_CFC_ (* Continuous Function Chart, elements in execution order *)
(* set timer cycle *)
(* delay on *)
(* delay off *)
#0 hw_reset_faults_id1 <= #1.DO1
#1 PLC:PLC110_32m2(FDI1: -, FDI2: -, DI1: hw_pressure_min, DI2: hw_pressure_max, DI3: ws_pressure_min, DI4: ws_pressure_max, DI5: hw_status_alarm_id1, DI6: hw_status_alarm_id2, DI7: ws_status_alarm_id1, DI8: ws_status_alarm_id2, DI9: hw_status_run_id1, DI10: hw_status_run_id2, DI11: ws_status_run_id1, DI12: ws_status_run_id2, DI13: -, DI14: -, DI15: -, DI16: -, SI: -, status_outputs: plc_outputs)
#2 ws_output_value_id2 <= #7.ch4_value
#3 analog_inputs_module:MB110_8a(ch1_error_code: hw_error_input_pressure, ch1_value: hw_input_pressure, ch2_error_code: hw_error_output_pressure, ch2_value: hw_output_pressure, ch3_error_code: ws_error_input_pressure, ch3_value: ws_input_pressure, ch4_error_code: ws_error_output_pressure, ch4_value: ws_output_pressure, ch5_error_code: -, ch5_value: -, ch6_error_code: -, ch6_value: -, ch7_error_code: -, ch7_value: -, ch8_error_code: -, ch8_value: -, settings: #20.settings)
#4 info_analog_inputs_module <= #3.info
#5 get_aout_current_in_info(info_invertor_drive: hw_info_id_1)
#6 currents_value_pack:get_info_analog_outputs_module(ch1_current: #5, ch2_current: #85, ch3_current: #86, ch4_current: #87, ch5_current: -, ch6_current: -, ch7_current: -, ch8_current: -)
#7 analog_outputs_module:MY110_8u(info_current_channel: #6.info)
#8 hw_run_id1 <= #1.FDO1
#9 get_run_in_info(info_invertor_drive: hw_info_id_1)
#10 PLC_110_32_outputs:get_status_outputs(fdo1: #9, fdo2: #15, fdo3: #79, fdo4: #81, do1: #16, do2: #111, do3: #112, do4: #113, do5: -, do6: -, do7: -, do8: -, do9: -, do10: -, do11: -, do12: -, do13: -, do14: -, do15: -, do16: -, sdo: -)
#11 plc_outputs <= #10.get_status_outputs
#12 hw_run_id2 <= #1.FDO2
#13 ws_run_id1 <= #1.FDO3
#14 ws_run_id2 <= #1.FDO4
#15 get_run_in_info(info_invertor_drive: hw_info_id_2)
#16 get_reset_faults(info: hw_info_id_1)
#17 value_scaling(input_value: hw_output_value_id1, params_scales: out_set_frequency)
#18 hw_frequency_id1 <= #17
#19 get_params_value_scaling(in_min: 0, in_max: 1000, out_min: 0, out_max: 50)
#20 settings_channel_analog_inputs_module:SetChannelsAnalogInputsModule(ch1_ain_l: -, ch1_ain_h: -, ch1_analog_min_value: -, ch1_analog_max_value: -, ch2_ain_l: -, ch2_ain_h: -, ch2_analog_min_value: -, ch2_analog_max_value: -, ch3_ain_l: -, ch3_ain_h: -, ch3_analog_min_value: -, ch3_analog_max_value: -, ch4_ain_l: -, ch4_ain_h: -, ch4_analog_min_value: -, ch4_analog_max_value: -, ch5_ain_l: -, ch5_ain_h: -, ch5_analog_min_value: -, ch5_analog_max_value: -, ch6_ain_l: -, ch6_ain_h: -, ch6_analog_min_value: -, ch6_analog_max_value: -, ch7_ain_l: -, ch7_ain_h: -, ch7_analog_min_value: -, ch7_analog_max_value: -, ch8_ain_l: -, ch8_ain_h: -, ch8_analog_min_value: -, ch8_analog_max_value: -)
#21 plc_inputs <= #1.status_inputs
#22 get_channel_current_value(ch_number: 1, Ain_info: info_analog_inputs_module)
#23 hw_input:CurrentSensorPressure_4_20(current_value: #22, set: -)
#24 hw_input_pressure_bar <= #23.pressure
#25 hw_settings_pressure_input:SetCurrentSensorPressure_4_20(min_measure_range: hw_min_measure_range_input, max_measure_range: hw_max_measure_range_input, min_current_range: -, max_current_range: -)
#26 get_channel_current_value(ch_number: 2, Ain_info: info_analog_inputs_module)
#27 hw_output:CurrentSensorPressure_4_20(current_value: #26, set: -)
#28 ws_input:CurrentSensorPressure_4_20(current_value: #108, set: -)
#29 ws_output:CurrentSensorPressure_4_20(current_value: #109, set: -)
#30 hw_output_pressure_bar <= #27.pressure
#31 hw_settings_pressure_output:SetCurrentSensorPressure_4_20(min_measure_range: hw_min_measure_range_output, max_measure_range: hw_max_measure_range_output, min_current_range: -, max_current_range: -)
#32 ws_input_pressure_bar <= #28.pressure
#33 ws_settings_pressure_input:SetCurrentSensorPressure_4_20(min_measure_range: ws_min_measure_range_input, max_measure_range: ws_max_measure_range_input, min_current_range: -, max_current_range: -)
#34 ws_output_pressure_bar <= #29.pressure
#35 ws_settings_pressure_output:SetCurrentSensorPressure_4_20(min_measure_range: ws_min_measure_range_output, max_measure_range: ws_max_measure_range_output, min_current_range: -, max_current_range: -)
#36 hw_kpi_35:Kpi(input: #37)
#37 get_di(input_number: 1, status_inputs: plc_inputs)
#38 hw_status_run_id1_sp <= #99
#39 hw_input_low_pressure_alarm <= #36.NO
#40 hw_invertor_drive_1:InvertorDrive(start: hw_start_id_1, reset_fault: hw_id1_reset_faults, low_pressure_in: #36.NO, high_pressure_out: #75.NO, status_run: #99, status_alarm: #46, ain_value: hw_output_pressure_bar, aout_value: hw_frequency_id_1, auto: hw_id1_auto, direct_logic: -, set_point: hw_set_point_pressure, P: -, I: -, D: -, manual: hw_manual_set_frequency_id1, min_range: -, max_range: -, active: hw_id1_active, system_alarm: hw_alarm_on)
#41 pid1:PID(#43.actual, #43.set_point, #43.P, #43.I, #43.D, #43.Y_manual, #43.Y_offset, #43.Y_min, #43.Y_max, #43.manual, #41.out 3)
#42 hw_info_id_1 <= #40.info
#43 hw_settings_pid_id_1:params_in_set_PID(set: #40.settings_pid)
#44 hw_frequency_id_1 <= #41.out 1
#45 get_di(input_number: 2, status_inputs: plc_inputs)
#46 get_di(input_number: 5, status_inputs: plc_inputs)
#47 hw_invertor_drive_2:InvertorDrive(start: hw_start_id_2, reset_fault: hw_id2_reset_faults, low_pressure_in: #36.NO, high_pressure_out: #75.NO, status_run: #101, status_alarm: #100, ain_value: hw_output_pressure_bar, aout_value: hw_frequency_id_2, auto: hw_id2_auto, direct_logic: -, set_point: hw_set_point_pressure, P: -, I: -, D: -, manual: hw_manual_set_frequency_id2, min_range: -, max_range: -, active: hw_id2_active, system_alarm: hw_alarm_on)
#48 pid2:PID(#49.actual, #49.set_point, #49.P, #49.I, #49.D, #49.Y_manual, #49.Y_offset, #49.Y_min, #49.Y_max, #49.manual, #48.out 3)
#49 hw_settings_pid_id_2:params_in_set_PID(set: #47.settings_pid)
#50 hw_frequency_id_2 <= #48.out 1
#51 get_di(input_number: 3, status_inputs: plc_inputs)
#52 hw_status_run_id2_sp <= #101
#53 ws_invertor_drive_1:InvertorDrive(start: ws_start_id_1, reset_fault: ws_id1_reset_faults, low_pressure_in: #58.NO, high_pressure_out: #76.NO, status_run: #104, status_alarm: #103, ain_value: ws_output_pressure_bar, aout_value: ws_frequency_id_1, auto: ws_id1_auto, direct_logic: -, set_point: ws_set_point_pressure, P: -, I: -, D: -, manual: ws_manual_set_frequency_id1, min_range: -, max_range: -, active: ws_id1_active, system_alarm: ws_alarm_on)
#54 pid3:PID(#56.actual, #56.set_point, #56.P, #56.I, #56.D, #56.Y_manual, #56.Y_offset, #56.Y_min, #56.Y_max, #56.manual, #54.out 3)
#55 ws_info_id_1 <= #53.info
#56 ws_settings_pid_id_1:params_in_set_PID(set: #53.settings_pid)
#57 ws_frequency_id_1 <= #54.out 1
#58 ws_kpi_35:Kpi(input: #51)
#59 ws_invertor_drive_2:InvertorDrive(start: ws_start_id_2, reset_fault: ws_id2_reset_faults, low_pressure_in: #58.NO, high_pressure_out: #76.NO, status_run: #107, status_alarm: #105, ain_value: ws_output_pressure_bar, aout_value: ws_frequency_id_2, auto: ws_id2_auto, direct_logic: -, set_point: ws_set_point_pressure, P: -, I: -, D: -, manual: ws_manual_set_frequency_id2, min_range: -, max_range: -, active: ws_id2_active, system_alarm: ws_alarm_on)
#60 pid4:PID(#62.actual, #62.set_point, #62.P, #62.I, #62.D, #62.Y_manual, #62.Y_offset, #62.Y_min, #62.Y_max, #62.manual, #60.out 3)
#61 ws_info_id_2 <= #59.info
#62 ws_settings_pid_id_2:params_in_set_PID(set: #59.settings_pid)
#63 ws_frequency_id_2 <= #60.out 1
#64 ws_status_run_id1_sp <= #104
#65 hw_single_mode:Single(enable: hw_single_enable, pivot_pump: hw_pivot_single, info_invertor_drive1: hw_info_id_1, info_invertor_drive2: hw_info_id_2, info_invertor_drive3: -, info_invertor_drive4: -, info_invertor_drive5: -, info_invertor_drive6: -, info_invertor_drive7: -, info_invertor_drive8: -)
#66 hw_mode_selector:Cascade_Cycle_Selector(cascade: hw_cascade_enable, cycle: hw_cycle_enable, single: hw_single_enable, info_single: #65.info_single, info_cycle: #69.info_cycle, info_cascade: #70.info_cascade)
#67 hw_start_id_1 <= #66.start_pump1
#68 hms_to_time(hours: hw_cycle_set_hours, minutes: hw_cycle_set_minutes, seconds: hw_cycle_set_seconds)
#69 hw_cycle_mode:cycle(enable: hw_cycle_enable, set_timer: #68, info_invertor_drive1: hw_info_id_1, info_invertor_drive2: hw_info_id_2, info_invertor_drive3: -, info_invertor_drive4: -, info_invertor_drive5: -, info_invertor_drive6: -, info_invertor_drive7: -, info_invertor_drive8: -)
#70 hw_cascade_mode:cascade(enable: hw_cascade_enable, set_pressure: hw_set_point_pressure, in_pressure: hw_input_pressure_bar, pivot_pump: hw_pivot_cascade, delay_on: #72, delay_off: #73, info_invertor_drive1: hw_info_id_1, info_invertor_drive2: hw_info_id_2, info_invertor_drive3: -, info_invertor_drive4: -, info_invertor_drive5: -, info_invertor_drive6: -, info_invertor_drive7: -, info_invertor_drive8: -)
#71 hw_start_id_2 <= #66.start_pump2
#72 hms_to_time(hours: hw_cascade_delay_on_hours, minutes: hw_cascade_delay_on_minutes, seconds: hw_cascade_delay_on_seconds)
#73 hms_to_time(hours: hw_cascade_delay_off_hours, minutes: hw_cascade_delay_off_minutes, seconds: hw_cascade_delay_off_seconds)
#74 hw_info_id_2 <= #47.info
#75 hw_kpi_36:Kpi(input: #45)
#76 ws_kpi_36:Kpi(input: #102)
#77 hw_reset_faults_id2 <= #1.DO2
#78 ws_reset_faults_id1 <= #1.DO3
#79 get_run_in_info(info_invertor_drive: ws_info_id_1)
#80 ws_reset_faults_id2 <= #1.DO4
#81 get_run_in_info(info_invertor_drive: ws_info_id_2)
#82 hw_output_value_id1 <= #7.ch1_value
#83 hw_output_value_id2 <= #7.ch2_value
#84 ws_output_value_id1 <= #7.ch3_value
#85 get_aout_current_in_info(info_invertor_drive: hw_info_id_2)
#86 get_aout_current_in_info(info_invertor_drive: ws_info_id_1)
#87 get_aout_current_in_info(info_invertor_drive: ws_info_id_2)
(* set timer cycle *)
(* delay on *)
(* delay off *)
#88 ws_single_mode:Single(enable: ws_single_enable, pivot_pump: ws_pivot_single, info_invertor_drive1: ws_info_id_1, info_invertor_drive2: ws_info_id_2, info_invertor_drive3: -, info_invertor_drive4: -, info_invertor_drive5: -, info_invertor_drive6: -, info_invertor_drive7: -, info_invertor_drive8: -)
#89 ws_mode_selector:Cascade_Cycle_Selector(cascade: ws_cascade_enable, cycle: ws_cycle_enable, single: ws_single_enable, info_single: #88.info_single, info_cycle: #93.info_cycle, info_cascade: #94.info_cascade)
#90 ws_start_id_1 <= #89.start_pump1
#91 hw_mode_error <= #66.mode_selector_error
#92 hms_to_time(hours: ws_cycle_set_hours, minutes: ws_cycle_set_minutes, seconds: ws_cycle_set_seconds)
#93 ws_cycle_mode:cycle(enable: ws_cycle_enable, set_timer: #92, info_invertor_drive1: ws_info_id_1, info_invertor_drive2: ws_info_id_2, info_invertor_drive3: -, info_invertor_drive4: -, info_invertor_drive5: -, info_invertor_drive6: -, info_invertor_drive7: -, info_invertor_drive8: -)
#94 ws_cascade_mode:cascade(enable: ws_cascade_enable, set_pressure: ws_set_point_pressure, in_pressure: ws_input_pressure_bar, pivot_pump: ws_pivot_cascade, delay_on: #97, delay_off: #98, info_invertor_drive1: ws_info_id_1, info_invertor_drive2: ws_info_id_2, info_invertor_drive3: -, info_invertor_drive4: -, info_invertor_drive5: -, info_invertor_drive6: -, info_invertor_drive7: -, info_invertor_drive8: -)
#95 ws_mode_error <= #89.mode_selector_error
#96 ws_start_id_2 <= #89.start_pump2
#97 hms_to_time(hours: ws_cascade_delay_on_hours, minutes: ws_cascade_delay_on_minutes, seconds: ws_cascade_delay_on_seconds)
#98 hms_to_time(hours: ws_cascade_delay_off_hours, minutes: ws_cascade_delay_off_minutes, seconds: ws_cascade_delay_off_seconds)
#99 get_di(input_number: 9, status_inputs: plc_inputs)
#100 get_di(input_number: 6, status_inputs: plc_inputs)
#101 get_di(input_number: 10, status_inputs: plc_inputs)
#102 get_di(input_number: 4, status_inputs: plc_inputs)
#103 get_di(input_number: 7, status_inputs: plc_inputs)
#104 get_di(input_number: 11, status_inputs: plc_inputs)
#105 get_di(input_number: 8, status_inputs: plc_inputs)
#106 ws_input_low_pressure_alarm <= #58.NO
#107 get_di(input_number: 12, status_inputs: plc_inputs)
#108 get_channel_current_value(ch_number: 3, Ain_info: info_analog_inputs_module)
#109 get_channel_current_value(ch_number: 4, Ain_info: info_analog_inputs_module)
#110 out_set_frequency <= #19
#111 get_reset_faults(info: hw_info_id_2)
#112 get_reset_faults(info: ws_info_id_1)
#113 get_reset_faults(info: ws_info_id_2)
#114 ws_status_run_id2_sp <= #107
#115 hw_out_high_pressure_alarm <= #75.NO
#116 ws_input_low_pressure_alarm <= #76.NO
#117 value_scaling(input_value: hw_output_value_id2, params_scales: out_set_frequency)
#118 hw_frequency_id2 <= #117
#119 value_scaling(input_value: ws_output_value_id1, params_scales: out_set_frequency)
#120 ws_frequency_id1 <= #119
#121 value_scaling(input_value: ws_output_value_id2, params_scales: out_set_frequency)
#122 ws_frequency_id2 <= #121
#123 get_di(input_number: 1, status_inputs: plc_inputs)
#124 get_di(input_number: 2, status_inputs: plc_inputs)
#125 hw_alarm_manager:ALARM_MANAGER(low_pressure_input: #123, high_pressure_out: #124, external_alarm_invertor_drive_code: #135.error_code_alarm, input_pressure_error_code: hw_error_input_pressure, out_pressure_error_code: hw_error_output_pressure, mode_selector_error: hw_mode_error)
#126 hw_alarm_on <= #125.alarm_on
#127 hw_alarm_error_code <= #125.error_code_alarm
#128 hw_alarm_message <= #125.error_message
#129 get_di(input_number: 3, status_inputs: plc_inputs)
#130 get_di(input_number: 4, status_inputs: plc_inputs)
#131 hw_alarm_manager:ALARM_MANAGER(low_pressure_input: #129, high_pressure_out: #130, external_alarm_invertor_drive_code: #136.error_code_alarm, input_pressure_error_code: ws_error_input_pressure, out_pressure_error_code: ws_error_output_pressure, mode_selector_error: ws_mode_error)
#132 ws_alarm_on <= #131.alarm_on
#133 ws_alarm_error_code <= #131.error_code_alarm
#134 ws_alarm_message <= #131.error_message
#135 hw_external_alarm:external_alarm_invertor_drive(status_inputs: plc_inputs, number_di_alarm_id1: 5, number_di_alarm_id2: 6, number_di_alarm_id3: -, number_di_alarm_id4: -, number_di_alarm_id5: -, number_di_alarm_id6: -, number_di_alarm_id7: -, number_di_alarm_id8: -)
#136 ws_external_alarm:external_alarm_invertor_drive(status_inputs: plc_inputs, number_di_alarm_id1: 7, number_di_alarm_id2: 8, number_di_alarm_id3: -, number_di_alarm_id4: -, number_di_alarm_id5: -, number_di_alarm_id6: -, number_di_alarm_id7: -, number_di_alarm_id8: -)
_END_CFC_
END_PROGRAM

(* POU PLC110_32/PLC110_32m2, ST *)
FUNCTION_BLOCK PLC110_32m2

VAR_INPUT
	FDI1:BOOL;
	FDI2:BOOL;
	DI1:BOOL;
	DI2:BOOL;
	DI3:BOOL;
	DI4:BOOL;
	DI5:BOOL;
	DI6:BOOL;
	DI7:BOOL;
	DI8:BOOL;
	DI9:BOOL;
	DI10:BOOL;
	DI11:BOOL;
	DI12:BOOL;
	DI13:BOOL;
	DI14:BOOL;
	DI15:BOOL;
	DI16:BOOL;
	SI:BOOL;
	status_outputs:classPLC32m2StatusOutputs;
END_VAR

VAR_OUTPUT
	FDO1:BOOL;
	FDO2:BOOL;
	FDO3:BOOL;
	FDO4:BOOL;
	DO1:BOOL;
	DO2:BOOL;
	DO3:BOOL;
	DO4:BOOL;
	DO5:BOOL;
	DO6:BOOL;
	DO7:BOOL;
	DO8:BOOL;
	DO9:BOOL;
	DO10:BOOL;
	DO11:BOOL;
	DO12:BOOL;
	DO13:BOOL;
	DO14:BOOL;
	DO15:BOOL;
	DO16:BOOL;
	SO:BOOL;
	status_inputs:classPLC32m2StatusInputs;
END_VAR

VAR
	fast_inputs:classFastDiscreteInputs;
	discrete_inputs:classDiscreteInputs;
	special_input:classSpecialInput;
	fast_outputs:classFastDiscreteOutputs;
	discrete_outputs:classDiscreteOutputs;
	special_output:classSpecialOutput;
END_VAR
init;

get_status_inputs;

get_status_outputs;
END_FUNCTION_BLOCK
ACTION get_status_inputs:
status_inputs.fast_inputs:=fast_inputs;
status_inputs.discrete_inputs:=discrete_inputs;
status_inputs.special_input:=special_input;
END_ACTION
ACTION get_status_outputs:
FDO1:=status_outputs.fast_outputs.Bit1;
FDO2:=status_outputs.fast_outputs.Bit2;
FDO3:=status_outputs.fast_outputs.Bit3;
FDO4:=status_outputs.fast_outputs.Bit4;

DO1:=status_outputs.discrete_outputs.first_byte.Bit1;
DO2:=status_outputs.discrete_outputs.first_byte.Bit2;
DO3:=status_outputs.discrete_outputs.first_byte.Bit3;
DO4:=status_outputs.discrete_outputs.first_byte.Bit4;
DO5:=status_outputs.discrete_outputs.first_byte.Bit5;
DO6:=status_outputs.discrete_outputs.first_byte.Bit6;
DO7:=status_outputs.discrete_outputs.first_byte.Bit7;
DO8:=status_outputs.discrete_outputs.first_byte.Bit8;
DO9:=status_outputs.discrete_outputs.second_byte.Bit1;
DO10:=status_outputs.discrete_outputs.second_byte.Bit2;
DO11:=status_outputs.discrete_outputs.second_byte.Bit3;
DO12:=status_outputs.discrete_outputs.second_byte.Bit4;
DO13:=status_outputs.discrete_outputs.second_byte.Bit5;
DO14:=status_outputs.discrete_outputs.second_byte.Bit6;
DO15:=status_outputs.discrete_outputs.second_byte.Bit7;
DO16:=status_outputs.discrete_outputs.second_byte.Bit8;

SO:=status_outputs.special_output.Bit1;
END_ACTION
ACTION init:
fast_inputs.Bit1:=FDI1;
fast_inputs.Bit2:=FDI2;

discrete_inputs.first_byte.Bit1:=DI1;
discrete_inputs.first_byte.Bit2:=DI2;
discrete_inputs.first_byte.Bit3:=DI3;
discrete_inputs.first_byte.Bit4:=DI4;
discrete_inputs.first_byte.Bit5:=DI5;
discrete_inputs.first_byte.Bit6:=DI6;
discrete_inputs.first_byte.Bit7:=DI7;
discrete_inputs.first_byte.Bit8:=DI8;
discrete_inputs.second_byte.Bit1:=DI9;
discrete_inputs.second_byte.Bit2:=DI10;
discrete_inputs.second_byte.Bit3:=DI11;
discrete_inputs.second_byte.Bit4:=DI12;
discrete_inputs.second_byte.Bit5:=DI13;
discrete_inputs.second_byte.Bit6:=DI14;
discrete_inputs.second_byte.Bit7:=DI15;
discrete_inputs.second_byte.Bit8:=DI16;

special_input.Bit1:=SI;

fast_outputs.Bit1:=FDO1;
fast_outputs.Bit2:=FDO2;
fast_outputs.Bit3:=FDO3;
fast_outputs.Bit4:=FDO4;

discrete_outputs.first_byte.Bit1:=DO1;
discrete_outputs.first_byte.Bit2:=DO2;
discrete_outputs.first_byte.Bit3:=DO3;
discrete_outputs.first_byte.Bit4:=DO4;
discrete_outputs.first_byte.Bit5:=DO5;
discrete_outputs.first_byte.Bit6:=DO6;
discrete_outputs.first_byte.Bit7:=DO7;
discrete_outputs.first_byte.Bit8:=DO8;

discrete_outputs.second_byte.Bit1:=DO9;
discrete_outputs.second_byte.Bit2:=DO10;
discrete_outputs.second_byte.Bit3:=DO11;
discrete_outputs.second_byte.Bit4:=DO12;
discrete_outputs.second_byte.Bit5:=DO13;
discrete_outputs.second_byte.Bit6:=DO14;
discrete_outputs.second_byte.Bit7:=DO15;
discrete_outputs.second_byte.Bit8:=DO16;

special_output.Bit1:=SO;
END_ACTION

(* POU PLC110_32/get_status_outputs, ST *)
FUNCTION_BLOCK get_status_outputs

VAR_INPUT
	fdo1:BOOL:=FALSE;
	fdo2:BOOL:=FALSE;
	fdo3:BOOL:=FALSE;
	fdo4:BOOL:=FALSE;
	do1:BOOL:=FALSE;
	do2:BOOL:=FALSE;
	do3:BOOL:=FALSE;
	do4:BOOL:=FALSE;
	do5:BOOL:=FALSE;
	do6:BOOL:=FALSE;
	do7:BOOL:=FALSE;
	do8:BOOL:=FALSE;
	do9:BOOL:=FALSE;
	do10:BOOL:=FALSE;
	do11:BOOL:=FALSE;
	do12:BOOL:=FALSE;
	do13:BOOL:=FALSE;
	do14:BOOL:=FALSE;
	do15:BOOL:=FALSE;
	do16:BOOL:=FALSE;
	sdo:BOOL:=FALSE;
END_VAR

VAR_OUTPUT
	get_status_outputs:classPLC32m2StatusOutputs;
END_VAR
get_status_outputs := get_status_outputs_def(fdo1, fdo2, fdo3, fdo4, do1, do2, do3, do4, do5, do6, do7, do8, do9, do10, do11, do12, do13, do14, do15, do16, sdo);
END_FUNCTION_BLOCK

(* POU PLC110_32/get_status_outputs_def, ST *)
FUNCTION get_status_outputs_def : classPLC32m2StatusOutputs

VAR_INPUT
	fdo1:BOOL:=FALSE;
	fdo2:BOOL:=FALSE;
	fdo3:BOOL:=FALSE;
	fdo4:BOOL:=FALSE;
	do1:BOOL:=FALSE;
	do2:BOOL:=FALSE;
	do3:BOOL:=FALSE;
	do4:BOOL:=FALSE;
	do5:BOOL:=FALSE;
	do6:BOOL:=FALSE;
	do7:BOOL:=FALSE;
	do8:BOOL:=FALSE;
	do9:BOOL:=FALSE;
	do10:BOOL:=FALSE;
	do11:BOOL:=FALSE;
	do12:BOOL:=FALSE;
	do13:BOOL:=FALSE;
	do14:BOOL:=FALSE;
	do15:BOOL:=FALSE;
	do16:BOOL:=FALSE;
	sdo:BOOL:=FALSE;
END_VAR
get_status_outputs_def.fast_outputs.Bit1:=fdo1;
get_status_outputs_def.fast_outputs.Bit2:=fdo2;
get_status_outputs_def.fast_outputs.Bit3:=fdo3;
get_status_outputs_def.fast_outputs.Bit4:=fdo4;

get_status_outputs_def.discrete_outputs.first_byte.Bit1:=do1;
get_status_outputs_def.discrete_outputs.first_byte.Bit2:=do2;
get_status_outputs_def.discrete_outputs.first_byte.Bit3:=do3;
get_status_outputs_def.discrete_outputs.first_byte.Bit4:=do4;
get_status_outputs_def.discrete_outputs.first_byte.Bit5:=do5;
get_status_outputs_def.discrete_outputs.first_byte.Bit6:=do6;
get_status_outputs_def.discrete_outputs.first_byte.Bit7:=do7;
get_status_outputs_def.discrete_outputs.first_byte.Bit8:=do8;
get_status_outputs_def.discrete_outputs.second_byte.Bit1:=do9;
get_status_outputs_def.discrete_outputs.second_byte.Bit2:=do10;
get_status_outputs_def.discrete_outputs.second_byte.Bit3:=do11;
get_status_outputs_def.discrete_outputs.second_byte.Bit4:=do12;
get_status_outputs_def.discrete_outputs.second_byte.Bit5:=do13;
get_status_outputs_def.discrete_outputs.second_byte.Bit6:=do14;
get_status_outputs_def.discrete_outputs.second_byte.Bit7:=do15;
get_status_outputs_def.discrete_outputs.second_byte.Bit8:=do16;

get_status_outputs_def.special_output.Bit1:=sdo;
END_FUNCTION

(* POU MB110_8.A/MB110_8a, ST *)
FUNCTION_BLOCK MB110_8a

VAR_INPUT
	ch1_error_code:WORD:=61447;
	ch1_value:REAL;
	ch2_error_code:WORD:=61447;
	ch2_value:REAL;
	ch3_error_code:WORD:=61447;
	ch3_value:REAL;
	ch4_error_code:WORD:=61447;
	ch4_value:REAL;
	ch5_error_code:WORD:=61447;
	ch5_value:REAL;
	ch6_error_code:WORD:=61447;
	ch6_value:REAL;
	ch7_error_code:WORD:=61447;
	ch7_value:REAL;
	ch8_error_code:WORD:=61447;
	ch8_value:REAL;
	settings:classSetAnalogInputsModule;
END_VAR

VAR_OUTPUT
	info:classInfoAnalogInputModule;
END_VAR
get_info_message;
END_FUNCTION_BLOCK
ACTION get_info_message:
info.channel1.error_message:=get_error_code(ch1_error_code);
info.channel2.error_message:=get_error_code(ch2_error_code);
info.channel3.error_message:=get_error_code(ch3_error_code);
info.channel4.error_message:=get_error_code(ch4_error_code);
info.channel5.error_message:=get_error_code(ch5_error_code);
info.channel6.error_message:=get_error_code(ch6_error_code);
info.channel7.error_message:=get_error_code(ch7_error_code);
info.channel8.error_message:=get_error_code(ch8_error_code);

info.channel1.current_value:=get_current_value(ch1_error_code,settings.ch1_set, ch1_value);
info.channel2.current_value:=get_current_value(ch2_error_code,settings.ch2_set, ch2_value);
info.channel3.current_value:=get_current_value(ch3_error_code,settings.ch3_set, ch3_value);
info.channel4.current_value:=get_current_value(ch4_error_code,settings.ch4_set, ch4_value);
info.channel5.current_value:=get_current_value(ch5_error_code,settings.ch5_set, ch5_value);
info.channel6.current_value:=get_current_value(ch6_error_code,settings.ch6_set, ch6_value);
info.channel7.current_value:=get_current_value(ch7_error_code,settings.ch7_set, ch7_value);
info.channel8.current_value:=get_current_value(ch8_error_code,settings.ch8_set, ch8_value);
END_ACTION

(* POU MB110_8.A/get_error_code, ST *)
FUNCTION get_error_code: STRING(79)
(* ï¿½ï¿½ï¿½ï¿½ï¿½ï¿½ï¿½ ï¿½ï¿½ï¿½ï¿½ï¿½ï¿½ï¿½ï¿½ï¿½ï¿½ï¿½ï¿½ï¿½ï¿½ ï¿½ï¿½ï¿½ï¿½ ï¿½ï¿½ï¿½ï¿½ï¿½ï¿½ ï¿½ï¿½ï¿½ï¿½ï¿½ï¿½ï¿½ï¿½ ï¿½ï¿½ï¿½ï¿½ï¿½ï¿½ï¿½ï¿½ï¿½ï¿½ï¿½ ï¿½ï¿½ï¿½ï¿½ï¿½ï¿½ ï¿½ï¿½ï¿½ï¿½ï¿½ï¿½ *)

VAR_INPUT
	code_error: WORD;
END_VAR

VAR
	error_message: STRING(79);
END_VAR
IF code_error=0
	THEN error_message := 'ï¿½ï¿½ï¿½ï¿½ï¿½ï¿½ï¿½ï¿½ï¿½ ï¿½ï¿½ï¿½ï¿½ï¿½ï¿½ï¿½';
ELSIF code_error = 61440
	THEN error_message := 'ï¿½ï¿½ï¿½ï¿½ï¿½ï¿½ï¿½ï¿½ ï¿½ï¿½ï¿½ï¿½ï¿½ï¿½ï¿½ï¿½ ï¿½ï¿½ï¿½ï¿½ï¿½ï¿½ï¿½';
ELSIF code_error = 61446
	THEN error_message := 'ï¿½ï¿½ï¿½ï¿½ï¿½ï¿½ ï¿½ï¿½ ï¿½ï¿½ï¿½ï¿½ï¿½ï¿½. ï¿½ï¿½ï¿½ï¿½ï¿½ ï¿½ï¿½ï¿½ï¿½ï¿½ï¿½ï¿½ï¿½ï¿½ï¿½ï¿½ ï¿½ï¿½ï¿½ï¿½ï¿½ï¿½ï¿½ ï¿½ï¿½ï¿½ï¿½ï¿½ï¿½ï¿½ï¿½ï¿½.';
ELSIF code_error = 61447
	THEN error_message := 'ï¿½ï¿½ï¿½ï¿½ï¿½ï¿½ ï¿½ï¿½ï¿½ï¿½ï¿½ï¿½ï¿½ï¿½.';
ELSIF code_error = 61448
	THEN error_message := 'ï¿½ï¿½ï¿½ï¿½ï¿½ï¿½ ï¿½ï¿½ï¿½ï¿½ï¿½ï¿½ï¿½ï¿½ï¿½ï¿½ï¿½ ï¿½ï¿½ï¿½ï¿½ï¿½ï¿½ï¿½ï¿½ï¿½ ï¿½ï¿½ï¿½ï¿½ï¿½ï¿½ ï¿½ï¿½.';
ELSIF code_error = 61449
	THEN error_message := 'ï¿½ï¿½ï¿½ï¿½ ï¿½ï¿½ï¿½ï¿½ï¿½ï¿½ï¿½ï¿½ï¿½ï¿½ï¿½ ï¿½ï¿½ï¿½ï¿½ï¿½ï¿½ï¿½ï¿½ï¿½ ï¿½ï¿½ï¿½ï¿½ï¿½ï¿½ ï¿½ï¿½.';
ELSIF code_error = 61450
	THEN error_message := 'ï¿½ï¿½ï¿½ï¿½ï¿½ï¿½ï¿½ï¿½ï¿½ï¿½ ï¿½ï¿½ï¿½ï¿½ï¿½ï¿½ï¿½ï¿½ ï¿½ï¿½ï¿½ï¿½ï¿½ï¿½ï¿½ ï¿½ï¿½ï¿½ï¿½ï¿½ï¿½.';
ELSIF code_error = 61451
	THEN error_message := 'ï¿½ï¿½ï¿½ï¿½ï¿½ï¿½ï¿½ï¿½ï¿½ï¿½ ï¿½ï¿½ï¿½ï¿½ï¿½ï¿½ï¿½ï¿½ ï¿½ï¿½ï¿½ï¿½ï¿½ï¿½ï¿½ ï¿½ï¿½ï¿½ï¿½.';
ELSIF code_error = 61452
	THEN error_message := 'ï¿½ï¿½ï¿½ï¿½ï¿½ï¿½ï¿½ï¿½ ï¿½ï¿½ï¿½ï¿½ï¿½ï¿½ï¿½ï¿½ï¿½ ï¿½ï¿½ï¿½ï¿½ï¿½ï¿½ï¿½.';
ELSIF code_error = 61453
	THEN error_message := 'ï¿½ï¿½ï¿½ï¿½ï¿½ ï¿½ï¿½ï¿½ï¿½ï¿½ï¿½ï¿½.';
ELSIF code_error = 61454
	THEN error_message := 'ï¿½ï¿½ï¿½ï¿½ï¿½ï¿½ï¿½ï¿½ï¿½ï¿½ ï¿½ï¿½ï¿½ï¿½ï¿½ ï¿½ ï¿½ï¿½ï¿½.';
ELSIF code_error = 61455
	THEN error_message := 'ï¿½ï¿½ï¿½ï¿½ï¿½ï¿½ï¿½ï¿½ï¿½ï¿½ï¿½ï¿½ ï¿½ï¿½ï¿½ï¿½ï¿½ï¿½ï¿½ï¿½ï¿½ï¿½ï¿½ï¿½ï¿½ ï¿½ï¿½ï¿½ï¿½ï¿½ï¿½ï¿½ï¿½ï¿½ï¿½ï¿½.';
ELSE
	error_message := 'Error not Found';
END_IF

get_error_code := error_message;
END_FUNCTION

(* POU MB110_8.A/get_current_value, ST *)
FUNCTION get_current_value : REAL
(* ï¿½ï¿½ï¿½ï¿½ï¿½ï¿½ï¿½ ï¿½ï¿½ï¿½ï¿½ï¿½ï¿½ï¿½ï¿½ï¿½ï¿½ï¿½ï¿½ï¿½ï¿½ï¿½ ï¿½ï¿½ï¿½ï¿½ï¿½ï¿½ ï¿½ ï¿½ï¿½ï¿½ ï¿½ ï¿½ï¿½ï¿½ï¿½ï¿½ï¿½ï¿½ï¿½ ï¿½ï¿½ï¿½ï¿½ *)

VAR_INPUT
	code_error:WORD;
	ch_set:classSetAnalogInputChannel;
	ch_value:REAL;
END_VAR
IF code_error = 0 THEN
	get_current_value := value_scaling(ch_value, get_set_Ain_value_params(ch_set));
ELSE
	(* ï¿½ï¿½ï¿½ï¿½ ï¿½ï¿½ï¿½ï¿½ï¿½ï¿½ ï¿½ï¿½ï¿½ï¿½ï¿½ï¿½ ï¿½ï¿½ï¿½ï¿½ï¿½ï¿½ ï¿½ï¿½ï¿½ï¿½ï¿½ï¿½ï¿½ ï¿½ï¿½ï¿½ï¿½ï¿½ï¿½ *)
	get_current_value := -8;
END_IF;
END_FUNCTION

(* POU function/value_scale/value_scaling, ST *)
FUNCTION value_scaling : REAL
(* ï¿½ï¿½ï¿½ï¿½ï¿½ï¿½ï¿½ ï¿½ï¿½ï¿½ï¿½ï¿½ï¿½ï¿½ï¿½ï¿½ï¿½ï¿½ï¿½ï¿½ï¿½ï¿½ ï¿½ï¿½ï¿½ï¿½ï¿½ *)

VAR_INPUT
	input_value: REAL;
	params_scales:classParamsValueScaling;
END_VAR

VAR
	A: REAL;
	B: REAL;
END_VAR
A := (params_scales.out_max - params_scales.out_min) / (params_scales.in_max - params_scales.in_min);
B := ((params_scales.out_min * params_scales.in_max) - (params_scales.out_max * params_scales.in_min)) / (params_scales.in_max - params_scales.in_min);

value_scaling := A * input_value + B;
END_FUNCTION

(* POU MB110_8.A/get_set_Ain_value_params, ST *)
FUNCTION get_set_Ain_value_params : classParamsValueScaling
(* ï¿½ï¿½ï¿½ï¿½ï¿½ï¿½ï¿½ï¿½ï¿½ï¿½ï¿½ï¿½ï¿½ï¿½ ï¿½ï¿½ ï¿½ï¿½ï¿½ï¿½ ï¿½ï¿½ï¿½ï¿½ï¿½ï¿½ï¿½ï¿½ ï¿½ï¿½ï¿½ï¿½ï¿½ ï¿½ ï¿½ï¿½ï¿½ï¿½ï¿½ï¿½ï¿½ï¿½ï¿½ ï¿½ï¿½ï¿½ï¿½ï¿½ï¿½ï¿½ï¿½ï¿½ï¿½ï¿½ï¿½ï¿½ï¿½ï¿½ *)

VAR_INPUT
	set:classSetAnalogInputChannel;
END_VAR
get_set_Ain_value_params.in_min:=set.ain_l;
get_set_Ain_value_params.in_max:=set.ain_h;
get_set_Ain_value_params.out_min:=set.analog_min_value;
get_set_Ain_value_params.out_max:=set.analog_max_value;
END_FUNCTION

(* POU MB110_8U/get_info_analog_outputs_module, ST *)
FUNCTION_BLOCK get_info_analog_outputs_module

VAR_INPUT
	ch1_current:REAL;
	ch2_current:REAL;
	ch3_current:REAL;
	ch4_current:REAL;
	ch5_current:REAL;
	ch6_current:REAL;
	ch7_current:REAL;
	ch8_current:REAL;
END_VAR

VAR_OUTPUT
	info:classAnalogOutputModule;
END_VAR
info.channel1.current_value := ch1_current;
info.channel2.current_value := ch2_current;
info.channel3.current_value := ch3_current;
info.channel4.current_value := ch4_current;
info.channel5.current_value := ch5_current;
info.channel6.current_value := ch6_current;
info.channel7.current_value := ch7_current;
info.channel8.current_value := ch8_current;
END_FUNCTION_BLOCK

(* POU MB110_8U/MY110_8u, ST *)
FUNCTION_BLOCK MY110_8u

VAR_INPUT
	info_current_channel:classAnalogOutputModule;
END_VAR

VAR_OUTPUT
	ch1_value:WORD;
	ch2_value:WORD;
	ch3_value:WORD;
	ch4_value:WORD;
	ch5_value:WORD;
	ch6_value:WORD;
	ch7_value:WORD;
	ch8_value:WORD;
END_VAR

VAR
	ch_ain_l: REAL := 4;  (* ï¿½ï¿½ï¿½ï¿½ï¿½ï¿½ï¿½ï¿½ ï¿½ï¿½ï¿½ï¿½ï¿½ï¿½ ï¿½ï¿½ï¿½ï¿½ï¿½ï¿½ï¿½ ï¿½ï¿½ï¿½ï¿½ï¿½ï¿½ï¿½ï¿½ ï¿½ï¿½ï¿½ï¿½ï¿½ï¿½ï¿½ï¿½ï¿½ *)
	ch_ain_h: REAL := 20;  (* ï¿½ï¿½ï¿½ï¿½ï¿½ï¿½ï¿½ï¿½ ï¿½ï¿½ï¿½ï¿½ï¿½ï¿½ï¿½ ï¿½ï¿½ï¿½ï¿½ï¿½ï¿½ï¿½ ï¿½ï¿½ï¿½ï¿½ï¿½ï¿½ï¿½ï¿½ ï¿½ï¿½ï¿½ï¿½ï¿½ï¿½ï¿½ï¿½ï¿½ *)
	ch_analog_min_value: REAL :=  0;  (* ï¿½ï¿½ï¿½ï¿½ï¿½ï¿½ ï¿½ï¿½ï¿½ï¿½ï¿½ï¿½ï¿½ ï¿½ï¿½ï¿½ *)
	ch_analog_max_value: REAL := 1000;  (* ï¿½ï¿½ï¿½ï¿½ï¿½ï¿½ï¿½ ï¿½ï¿½ï¿½ï¿½ï¿½ï¿½ï¿½ ï¿½ï¿½ï¿½ *)
	set_params:classParamsValueScaling;
END_VAR
set_params := get_params_value_scaling(ch_ain_l, ch_ain_h, ch_analog_min_value, ch_analog_max_value);

ch1_value := REAL_TO_INT(value_scaling(info_current_channel.channel1.current_value, set_params));
ch2_value := REAL_TO_INT(value_scaling(info_current_channel.channel2.current_value, set_params));
ch3_value := REAL_TO_INT(value_scaling(info_current_channel.channel3.current_value, set_params));
ch4_value := REAL_TO_INT(value_scaling(info_current_channel.channel4.current_value, set_params));
ch5_value := REAL_TO_INT(value_scaling(info_current_channel.channel5.current_value, set_params));
ch6_value := REAL_TO_INT(value_scaling(info_current_channel.channel6.current_value, set_params));
ch7_value := REAL_TO_INT(value_scaling(info_current_channel.channel7.current_value, set_params));
ch8_value := REAL_TO_INT(value_scaling(info_current_channel.channel8.current_value, set_params));
END_FUNCTION_BLOCK

(* POU function/value_scale/get_params_value_scaling, ST *)
FUNCTION get_params_value_scaling : classParamsValueScaling

VAR_INPUT
	in_min: REAL;
	in_max: REAL;
	out_min: REAL;
	out_max: REAL;
END_VAR
get_params_value_scaling.in_min := in_min;
get_params_value_scaling.in_max := in_max;
get_params_value_scaling.out_min := out_min;
get_params_value_scaling.out_max := out_max;
END_FUNCTION

(* POU MB110_8.A/SetChannelsAnalogInputsModule, ST *)
FUNCTION_BLOCK SetChannelsAnalogInputsModule

VAR_INPUT
	(* ï¿½ï¿½ï¿½ï¿½ï¿½ï¿½ï¿½ï¿½ï¿½ï¿½ï¿½ï¿½ï¿½ï¿½ï¿½ï¿½ ï¿½ï¿½ï¿½ï¿½ï¿½ï¿½ï¿½ï¿½ï¿½ ï¿½ï¿½ï¿½ï¿½ï¿½ï¿½ ï¿½ï¿½ï¿½ï¿½ï¿½ï¿½. ï¿½ï¿½. ï¿½ï¿½ï¿½ï¿½ï¿½ï¿½ï¿½ï¿½ï¿½ï¿½ ï¿½ï¿½ï¿½ï¿½ï¿½ï¿½ï¿½: ï¿½ï¿½ï¿½ï¿½ï¿½ï¿½ï¿½ï¿½ï¿½ï¿½. ï¿½ï¿½ï¿½ï¿½ï¿½ï¿½ï¿½ ï¿½.2 *)
	(* ï¿½ï¿½ï¿½ï¿½ï¿½ï¿½ï¿½ ï¿½ï¿½ï¿½ ï¿½ ï¿½ï¿½ï¿½ï¿½ï¿½ï¿½ï¿½ï¿½ ï¿½ï¿½ ï¿½ï¿½ï¿½ï¿½ï¿½ï¿½ï¿½ï¿½ï¿½: ï¿½ï¿½ï¿½ ï¿½ï¿½ï¿½ï¿½ï¿½ï¿½ï¿½ 4-20mA  *)

	ch1_ain_l: REAL := 0;  (* ï¿½ï¿½ï¿½ï¿½ï¿½ï¿½ï¿½ï¿½ Ain.L *)
	ch1_ain_h: REAL := 100;  (* ï¿½ï¿½ï¿½ï¿½ï¿½ï¿½ï¿½ï¿½ Ain.H *)
	ch1_analog_min_value: REAL := 4;  (* ï¿½ï¿½ï¿½ï¿½ï¿½ï¿½ï¿½ï¿½ ï¿½ï¿½ï¿½ï¿½ï¿½ï¿½ ï¿½ï¿½ï¿½ï¿½ï¿½ï¿½ï¿½ ï¿½ï¿½ï¿½ï¿½ï¿½ï¿½ï¿½ *)
	ch1_analog_max_value: REAL := 20;  (* ï¿½ï¿½ï¿½ï¿½ï¿½ï¿½ï¿½ï¿½ ï¿½ï¿½ï¿½ï¿½ï¿½ï¿½ï¿½ ï¿½ï¿½ï¿½ï¿½ï¿½ï¿½ï¿½ ï¿½ï¿½ï¿½ï¿½ï¿½ï¿½ï¿½ *)

	ch2_ain_l: REAL := 0;  (* ï¿½ï¿½ï¿½ï¿½ï¿½ï¿½ï¿½ï¿½ Ain.L *)
	ch2_ain_h: REAL := 100;  (* ï¿½ï¿½ï¿½ï¿½ï¿½ï¿½ï¿½ï¿½ Ain.H *)
	ch2_analog_min_value: REAL := 4;  (* ï¿½ï¿½ï¿½ï¿½ï¿½ï¿½ï¿½ï¿½ ï¿½ï¿½ï¿½ï¿½ï¿½ï¿½ ï¿½ï¿½ï¿½ï¿½ï¿½ï¿½ï¿½ ï¿½ï¿½ï¿½ï¿½ï¿½ï¿½ï¿½ *)
	ch2_analog_max_value: REAL := 20;  (* ï¿½ï¿½ï¿½ï¿½ï¿½ï¿½ï¿½ï¿½ ï¿½ï¿½ï¿½ï¿½ï¿½ï¿½ï¿½ ï¿½ï¿½ï¿½ï¿½ï¿½ï¿½ï¿½ ï¿½ï¿½ï¿½ï¿½ï¿½ï¿½ï¿½ *)

	ch3_ain_l: REAL := 0;  (* ï¿½ï¿½ï¿½ï¿½ï¿½ï¿½ï¿½ï¿½ Ain.L *)
	ch3_ain_h: REAL := 100;  (* ï¿½ï¿½ï¿½ï¿½ï¿½ï¿½ï¿½ï¿½ Ain.H *)
	ch3_analog_min_value: REAL := 4;  (* ï¿½ï¿½ï¿½ï¿½ï¿½ï¿½ï¿½ï¿½ ï¿½ï¿½ï¿½ï¿½ï¿½ï¿½ ï¿½ï¿½ï¿½ï¿½ï¿½ï¿½ï¿½ ï¿½ï¿½ï¿½ï¿½ï¿½ï¿½ï¿½ *)
	ch3_analog_max_value: REAL := 20;  (* ï¿½ï¿½ï¿½ï¿½ï¿½ï¿½ï¿½ï¿½ ï¿½ï¿½ï¿½ï¿½ï¿½ï¿½ï¿½ ï¿½ï¿½ï¿½ï¿½ï¿½ï¿½ï¿½ ï¿½ï¿½ï¿½ï¿½ï¿½ï¿½ï¿½ *)

	ch4_ain_l: REAL := 0;  (* ï¿½ï¿½ï¿½ï¿½ï¿½ï¿½ï¿½ï¿½ Ain.L *)
	ch4_ain_h: REAL := 100;  (* ï¿½ï¿½ï¿½ï¿½ï¿½ï¿½ï¿½ï¿½ Ain.H *)
	ch4_analog_min_value: REAL := 4;  (* ï¿½ï¿½ï¿½ï¿½ï¿½ï¿½ï¿½ï¿½ ï¿½ï¿½ï¿½ï¿½ï¿½ï¿½ ï¿½ï¿½ï¿½ï¿½ï¿½ï¿½ï¿½ ï¿½ï¿½ï¿½ï¿½ï¿½ï¿½ï¿½ *)
	ch4_analog_max_value: REAL := 20;  (* ï¿½ï¿½ï¿½ï¿½ï¿½ï¿½ï¿½ï¿½ ï¿½ï¿½ï¿½ï¿½ï¿½ï¿½ï¿½ ï¿½ï¿½ï¿½ï¿½ï¿½ï¿½ï¿½ ï¿½ï¿½ï¿½ï¿½ï¿½ï¿½ï¿½ *)

	ch5_ain_l: REAL := 0;  (* ï¿½ï¿½ï¿½ï¿½ï¿½ï¿½ï¿½ï¿½ Ain.L *)
	ch5_ain_h: REAL := 100;  (* ï¿½ï¿½ï¿½ï¿½ï¿½ï¿½ï¿½ï¿½ Ain.H *)
	ch5_analog_min_value: REAL := 4;  (* ï¿½ï¿½ï¿½ï¿½ï¿½ï¿½ï¿½ï¿½ ï¿½ï¿½ï¿½ï¿½ï¿½ï¿½ ï¿½ï¿½ï¿½ï¿½ï¿½ï¿½ï¿½ ï¿½ï¿½ï¿½ï¿½ï¿½ï¿½ï¿½ *)
	ch5_analog_max_value: REAL := 20;  (* ï¿½ï¿½ï¿½ï¿½ï¿½ï¿½ï¿½ï¿½ ï¿½ï¿½ï¿½ï¿½ï¿½ï¿½ï¿½ ï¿½ï¿½ï¿½ï¿½ï¿½ï¿½ï¿½ ï¿½ï¿½ï¿½ï¿½ï¿½ï¿½ï¿½ *)

	ch6_ain_l: REAL := 0;  (* ï¿½ï¿½ï¿½ï¿½ï¿½ï¿½ï¿½ï¿½ Ain.L *)
	ch6_ain_h: REAL := 100;  (* ï¿½ï¿½ï¿½ï¿½ï¿½ï¿½ï¿½ï¿½ Ain.H *)
	ch6_analog_min_value: REAL := 4;  (* ï¿½ï¿½ï¿½ï¿½ï¿½ï¿½ï¿½ï¿½ ï¿½ï¿½ï¿½ï¿½ï¿½ï¿½ ï¿½ï¿½ï¿½ï¿½ï¿½ï¿½ï¿½ ï¿½ï¿½ï¿½ï¿½ï¿½ï¿½ï¿½ *)
	ch6_analog_max_value: REAL := 20;  (* ï¿½ï¿½ï¿½ï¿½ï¿½ï¿½ï¿½ï¿½ ï¿½ï¿½ï¿½ï¿½ï¿½ï¿½ï¿½ ï¿½ï¿½ï¿½ï¿½ï¿½ï¿½ï¿½ ï¿½ï¿½ï¿½ï¿½ï¿½ï¿½ï¿½ *)

	ch7_ain_l: REAL := 0;  (* ï¿½ï¿½ï¿½ï¿½ï¿½ï¿½ï¿½ï¿½ Ain.L *)
	ch7_ain_h: REAL := 100;  (* ï¿½ï¿½ï¿½ï¿½ï¿½ï¿½ï¿½ï¿½ Ain.H *)
	ch7_analog_min_value: REAL := 4;  (* ï¿½ï¿½ï¿½ï¿½ï¿½ï¿½ï¿½ï¿½ ï¿½ï¿½ï¿½ï¿½ï¿½ï¿½ ï¿½ï¿½ï¿½ï¿½ï¿½ï¿½ï¿½ ï¿½ï¿½ï¿½ï¿½ï¿½ï¿½ï¿½ *)
	ch7_analog_max_value: REAL := 20;  (* ï¿½ï¿½ï¿½ï¿½ï¿½ï¿½ï¿½ï¿½ ï¿½ï¿½ï¿½ï¿½ï¿½ï¿½ï¿½ ï¿½ï¿½ï¿½ï¿½ï¿½ï¿½ï¿½ ï¿½ï¿½ï¿½ï¿½ï¿½ï¿½ï¿½ *)

	ch8_ain_l: REAL := 0;  (* ï¿½ï¿½ï¿½ï¿½ï¿½ï¿½ï¿½ï¿½ Ain.L *)
	ch8_ain_h: REAL := 100;  (* ï¿½ï¿½ï¿½ï¿½ï¿½ï¿½ï¿½ï¿½ Ain.H *)
	ch8_analog_min_value: REAL := 4;  (* ï¿½ï¿½ï¿½ï¿½ï¿½ï¿½ï¿½ï¿½ ï¿½ï¿½ï¿½ï¿½ï¿½ï¿½ ï¿½ï¿½ï¿½ï¿½ï¿½ï¿½ï¿½ ï¿½ï¿½ï¿½ï¿½ï¿½ï¿½ï¿½ *)
	ch8_analog_max_value: REAL := 20;  (* ï¿½ï¿½ï¿½ï¿½ï¿½ï¿½ï¿½ï¿½ ï¿½ï¿½ï¿½ï¿½ï¿½ï¿½ï¿½ ï¿½ï¿½ï¿½ï¿½ï¿½ï¿½ï¿½ ï¿½ï¿½ï¿½ï¿½ï¿½ï¿½ï¿½ *)
END_VAR

VAR_OUTPUT
	settings:classSetAnalogInputsModule;
END_VAR
get_settings;
END_FUNCTION_BLOCK
ACTION get_settings:
settings.ch1_set := get_setAin(ch1_ain_l, ch1_ain_h, ch1_analog_min_value, ch1_analog_max_value);
settings.ch2_set := get_setAin(ch2_ain_l, ch2_ain_h, ch2_analog_min_value, ch2_analog_max_value);
settings.ch3_set := get_setAin(ch3_ain_l, ch3_ain_h, ch3_analog_min_value, ch3_analog_max_value);
settings.ch4_set := get_setAin(ch4_ain_l, ch4_ain_h, ch4_analog_min_value, ch4_analog_max_value);
settings.ch5_set := get_setAin(ch5_ain_l, ch5_ain_h, ch5_analog_min_value, ch5_analog_max_value);
settings.ch6_set := get_setAin(ch6_ain_l, ch6_ain_h, ch6_analog_min_value, ch6_analog_max_value);
settings.ch7_set := get_setAin(ch7_ain_l, ch7_ain_h, ch7_analog_min_value, ch7_analog_max_value);
settings.ch8_set := get_setAin(ch8_ain_l, ch8_ain_h, ch8_analog_min_value, ch8_analog_max_value);
END_ACTION

(* POU MB110_8.A/get_setAin, ST *)
FUNCTION get_setAin : classSetAnalogInputChannel
(* ï¿½ï¿½ï¿½ï¿½ï¿½ï¿½ï¿½ï¿½ï¿½ ï¿½ï¿½ï¿½ï¿½ï¿½ï¿½ï¿½ï¿½ ï¿½ dataclass *)

VAR_INPUT
	ch_ain_l: REAL := 0;  (* ï¿½ï¿½ï¿½ï¿½ï¿½ï¿½ï¿½ï¿½ Ain.L *)
	ch_ain_h: REAL := 100;  (* ï¿½ï¿½ï¿½ï¿½ï¿½ï¿½ï¿½ï¿½ Ain.H *)
	ch_analog_min_value: REAL := 4;  (* ï¿½ï¿½ï¿½ï¿½ï¿½ï¿½ï¿½ï¿½ ï¿½ï¿½ï¿½ï¿½ï¿½ï¿½ ï¿½ï¿½ï¿½ï¿½ï¿½ï¿½ï¿½ ï¿½ï¿½ï¿½ï¿½ï¿½ï¿½ï¿½ *)
	ch_analog_max_value: REAL := 20;  (* ï¿½ï¿½ï¿½ï¿½ï¿½ï¿½ï¿½ï¿½ ï¿½ï¿½ï¿½ï¿½ï¿½ï¿½ï¿½ ï¿½ï¿½ï¿½ï¿½ï¿½ï¿½ï¿½ ï¿½ï¿½ï¿½ï¿½ï¿½ï¿½ï¿½ *)
END_VAR
get_setAin.ain_l:=ch_ain_l;
get_setAin.ain_h:=ch_ain_h;
get_setAin.analog_min_value:=ch_analog_min_value;
get_setAin.analog_max_value:=ch_analog_max_value;
END_FUNCTION

(* POU PressureSensor_4_20ma/CurrentSensorPressure_4_20, ST *)
FUNCTION_BLOCK CurrentSensorPressure_4_20

VAR_INPUT
	current_value:REAL;  (*ï¿½ï¿½ï¿½ï¿½ï¿½ï¿½ï¿½ï¿½ ï¿½ï¿½ï¿½ï¿½ 4-20ï¿½ï¿½ *)
	set:classSetPressureSensor4_20;  (* ï¿½ï¿½ï¿½ï¿½ï¿½ï¿½ï¿½ ï¿½ ï¿½ï¿½ï¿½ï¿½ï¿½ï¿½ ï¿½ï¿½ï¿½ï¿½ï¿½ï¿½ï¿½ ï¿½ï¿½ï¿½ï¿½ï¿½ï¿½ï¿½ï¿½ *)
END_VAR

VAR_OUTPUT
	pressure:REAL;  (* ï¿½ï¿½ï¿½ï¿½ï¿½ï¿½ï¿½ï¿½ ï¿½ï¿½ ï¿½ï¿½ï¿½ï¿½ï¿½ï¿½ *)
END_VAR
pressure:=value_scaling(current_value, get_set_sensor_value_params(set));
END_FUNCTION_BLOCK

(* POU PressureSensor_4_20ma/get_set_sensor_value_params, ST *)
FUNCTION get_set_sensor_value_params : classParamsValueScaling

VAR_INPUT
	sensor_set:classSetPressureSensor4_20;
END_VAR
get_set_sensor_value_params.in_min := sensor_set.min_current_range;
get_set_sensor_value_params.in_max := sensor_set.max_current_range;
get_set_sensor_value_params.out_min := sensor_set.min_measure_range;
get_set_sensor_value_params.out_max := sensor_set.max_measure_range;
END_FUNCTION

(* POU Invertor_Drive/InvertorDrive, ST *)
FUNCTION_BLOCK InvertorDrive
(* Function block implementation invertor drive. *)

VAR_INPUT
(* discrete inputs *)
	start: BOOL := FALSE;
	reset_fault: BOOL := FALSE;
	low_pressure_in: BOOL;  (* external alarm *)
	high_pressure_out: BOOL;  (* external alrm *)
(* discrete outputs *)
	status_run: BOOL;
	status_alarm: BOOL;
(* analog inputs *)
	ain_value: REAL := 0;  (* mA or V *)
(* analog outputs *)
	aout_value: REAL := 0;
(* PID settings *)
	auto: BOOL := FALSE;
	direct_logic: BOOL := TRUE;  (* flag forward/reverse control, reverse control: if input value less set point, output value to less. forward control: if input value less set point, output value to more. *)
	set_point: REAL := 0;  (* set point, measure system in input value control. *)
	P: REAL := 2;  (* proporcional value of PID, if more, out value fasted. *)
	I: INT := 10;  (* integral value of PID, seconds *)
	D:INT := 0;  (* differential value PID, seconds *)

(* limit work frequency *)
	manual: REAL := 0; (* set output value in manual mode, Hz*)
	min_range: REAL := 15;  (* min value in manual mode, Hz*)
	max_range: REAL := 50;  (* max value in manual mode, Hz*)

(* status invertor in work *)
	active: BOOL := FALSE;  (* statis active invertor drive. *)
	system_alarm: BOOL; (* alarm manager alarm_on *)
END_VAR

VAR_OUTPUT
	info: classInfoInvertorDrive;
	settings_pid: classSetPid;
END_VAR

VAR
	invertor_drive: classInvertorDrive;
    set_auto: classSetAutoInvertorDrive;
	set_frequency: classSetLimitFrequency;
	set_pid: classSetPid;

	discrete_inputs: classInvertorDriveDiscreteInputs;
	discrete_outputs: classInvertorDriveDiscreteOutputs;
	analog_inputs: classInvertorDriveAnalogInputs;
	analog_outputs: classInvertorDriveAnalogOutputs;

	overflow: BOOL := FALSE; (* overflow integral value of PID *)

	external_alarm:STRING(79); (* message of external alarm. *)

	info_alarm: classAlarmInvertorDrive;
END_VAR
init;

info_alarm.external_alarm := get_external_alarm(
	discrete_inputs.low_pressure_in, discrete_inputs.high_pressure_out
);

get_PID_set;

get_infomessage;
END_FUNCTION_BLOCK
ACTION get_infoMessage:
info.active := active;
info.set_pid := set_pid;
info.alarm.external_alarm := info_alarm.external_alarm;

IF discrete_outputs.status_alarm THEN
	info_alarm.fault_invertor_drive := 'Alarm invertor drive!';
	analog_outputs.out_frequency := 0;
ELSE
	info_alarm.fault_invertor_drive := 'No alarm';
END_IF;

info.alarm.fault_invertor_drive := info_alarm.fault_invertor_drive;

IF discrete_outputs.status_run THEN
	info.status_run := 'Run';

ELSE
	info.status_run := 'Stopped';
	analog_outputs.out_frequency := 0;
END_IF;

(* converted frequency in current value of 4-20 mA *)
info.frequency := analog_outputs.out_frequency;
info.aout_frequency := value_scaling(analog_outputs.out_frequency, get_params_value_scaling(0, 50, 4, 20));

IF info.alarm.external_alarm  <> 'GOOD' THEN
	discrete_inputs.start := FALSE;
ELSIF info.alarm.fault_invertor_drive <> 'No alarm' THEN
	discrete_inputs.start := FALSE;
ELSIF system_alarm <> 0 THEN
	discrete_inputs.start := FALSE;
ELSE
	discrete_inputs.start := invertor_drive.discrete_inputs.start;
END_IF;

info.reset_fault := discrete_inputs.reset_fault;

info.run := discrete_inputs.start;
END_ACTION
ACTION get_PID_set:
analog_inputs := invertor_drive.analog_input;
set_auto := invertor_drive.set.set_auto;
set_frequency := invertor_drive.set.set_frequency;

overflow := FALSE; (* this place for realise reset integral value of PID *) 

set_pid := get_set_pid(
	set_auto.direct_logic,
	set_auto.value,
	set_auto.set_point,
	set_auto.P,
	set_auto.I,
	set_auto.D,
	set_frequency.manual,
	0,
	set_frequency.min_range,
	set_frequency.max_range,
	NOT set_auto.auto,
	overflow
);

settings_pid := set_pid;
END_ACTION
ACTION init:
invertor_drive.analog_input.set_frequency := ain_value;
invertor_drive.analog_output.out_frequency := aout_value;

invertor_drive.discrete_inputs.start := start;
invertor_drive.discrete_inputs.reset_fault := reset_fault;
invertor_drive.discrete_inputs.low_pressure_in := low_pressure_in;
invertor_drive.discrete_inputs.high_pressure_out := high_pressure_out;

invertor_drive.discrete_outputs.status_run := status_run;
invertor_drive.discrete_outputs.status_alarm := status_alarm;

invertor_drive.set.set_frequency.min_range := min_range;
invertor_drive.set.set_frequency.max_range := max_range;

invertor_drive.set.set_auto.auto := auto;
invertor_drive.set.set_auto.direct_logic := direct_logic;
invertor_drive.set.set_auto.set_point := set_point;
invertor_drive.set.set_auto.value := ain_value;
invertor_drive.set.set_auto.P := P;
invertor_drive.set.set_auto.I := I;
invertor_drive.set.set_auto.D := D;

invertor_drive.set.set_frequency.manual := manual;
invertor_drive.set.set_frequency.min_range := min_range;
invertor_drive.set.set_frequency.max_range := max_range;

discrete_inputs := invertor_drive.discrete_inputs;
discrete_outputs := invertor_drive.discrete_outputs;
analog_outputs := invertor_drive.analog_output;
END_ACTION

(* POU Invertor_Drive/get_external_alarm, ST *)
FUNCTION get_external_alarm : STRING(79)
(* ï¿½ï¿½ï¿½ï¿½ï¿½ï¿½ï¿½ï¿½ï¿½ ï¿½ï¿½ï¿½ï¿½ï¿½ï¿½ï¿½ï¿½ï¿½ ï¿½ï¿½ï¿½ï¿½ï¿½ï¿½ ï¿½ï¿½ ï¿½ï¿½ï¿½ï¿½ï¿½ï¿½ ï¿½ï¿½ï¿½ï¿½ ï¿½ï¿½ï¿½ ï¿½ï¿½ï¿½ï¿½ï¿½ï¿½ï¿½ï¿½ï¿½ï¿½ ï¿½ï¿½ï¿½ï¿½ï¿½ï¿½ï¿½ï¿½ *)
VAR_INPUT
	low_pressure_in:BOOL;
	high_pressure_out:BOOL;
END_VAR
IF low_pressure_in THEN
	get_external_alarm:='ï¿½ï¿½ï¿½ï¿½ï¿½ï¿½ ï¿½ï¿½ï¿½ï¿½ï¿½ï¿½ï¿½ï¿½ ï¿½ï¿½ ï¿½ï¿½ï¿½ï¿½ï¿½';
ELSIF high_pressure_out THEN
	get_external_alarm:='ï¿½ï¿½ï¿½ï¿½ï¿½ï¿½ï¿½ ï¿½ï¿½ï¿½ï¿½ï¿½ï¿½ï¿½ï¿½ ï¿½ï¿½ ï¿½ï¿½ï¿½ï¿½ï¿½ï¿½';
ELSE
	get_external_alarm:='GOOD';
END_IF;
END_FUNCTION

(* POU PID_regulator/get_set_pid, ST *)
FUNCTION get_set_pid : classSetPid

VAR_INPUT
	direct_logic:BOOL:=TRUE;
	actual:REAL;
	set_point:REAL;
	P:REAL:=2;  (* ï¿½ï¿½ï¿½ï¿½ï¿½ï¿½ï¿½ï¿½ï¿½ï¿½ï¿½ï¿½ï¿½ï¿½ï¿½ï¿½ ï¿½ï¿½ï¿½ï¿½ï¿½ï¿½ï¿½ï¿½ï¿½ï¿½ï¿½ ï¿½ï¿½ï¿½ï¿½ï¿½ï¿½ï¿½ï¿½ï¿½ï¿½, ï¿½ï¿½ï¿½ ï¿½ï¿½ï¿½ï¿½ï¿½ï¿½ï¿½ï¿½ï¿½ï¿½ ï¿½ï¿½ï¿½ï¿½ï¿½ ï¿½ï¿½ï¿½ï¿½ï¿½ï¿½ï¿½ï¿½ï¿½ï¿½ ï¿½ï¿½ï¿½ï¿½ï¿½ï¿½ï¿½ï¿½ï¿½ï¿½ ï¿½ï¿½ï¿½ï¿½ï¿½ï¿½ï¿½*)
	I:INT:=10;  (* ï¿½ï¿½ï¿½ï¿½ï¿½ï¿½ï¿½ï¿½ï¿½ï¿½ï¿½ï¿½ ï¿½ï¿½ï¿½ï¿½ï¿½ï¿½ï¿½ï¿½ï¿½ï¿½ï¿½ ï¿½ï¿½ï¿½ï¿½ï¿½ï¿½ï¿½ï¿½ï¿½ï¿½, ï¿½ï¿½ï¿½ï¿½ï¿½ ï¿½ ï¿½ï¿½ï¿½ï¿½ï¿½ï¿½ï¿½ï¿½ *)
	D:INT:=0;  (* ï¿½ï¿½ï¿½ï¿½ï¿½ï¿½ï¿½ï¿½ï¿½ï¿½ï¿½ï¿½ï¿½ï¿½ï¿½ï¿½ ï¿½ï¿½ï¿½ï¿½ï¿½ï¿½ï¿½ï¿½ï¿½ï¿½ï¿½ ï¿½ï¿½ï¿½ï¿½ï¿½ï¿½ï¿½ï¿½ï¿½ï¿½, ï¿½ï¿½ï¿½ï¿½ï¿½ ï¿½ ï¿½ï¿½ï¿½ï¿½ï¿½ï¿½ï¿½ï¿½ *)
	Y_manual:REAL:=0;  (* Hz *)
	Y_offset:REAL:=0;
	Y_min:REAL;
	Y_max:REAL;
	manual:BOOL:=TRUE;  (* ï¿½ï¿½ï¿½ï¿½ï¿½ï¿½ï¿½ï¿½ï¿½ï¿½ï¿½ ï¿½ï¿½ï¿½ï¿½ï¿½ï¿½ï¿½ï¿½ ï¿½ï¿½ï¿½ï¿½ï¿½ï¿½ ï¿½ï¿½ï¿½ï¿½ï¿½ *)
	reset:BOOL:=FALSE;
END_VAR
IF direct_logic = TRUE THEN
	get_set_pid.actual := actual;
	get_set_pid.set_point := set_point;
ELSE
	get_set_pid.actual := set_point;
	get_set_pid.set_point := actual;
END_IF;

get_set_pid.P := P;
get_set_pid.I := I;
get_set_pid.D := D;
get_set_pid.Y_manual := Y_manual;
get_set_pid.Y_offset := Y_offset;
get_set_pid.Y_min := Y_min;
get_set_pid.Y_max := Y_max;
get_set_pid.manual := manual;
get_set_pid.reset := reset;
END_FUNCTION

(* POU PID_regulator/params_in_set_PID, ST *)
FUNCTION_BLOCK params_in_set_PID

VAR_INPUT
	set:classSetPid;
END_VAR

VAR_OUTPUT
	actual:REAL;
	set_point:REAL;
	P:REAL;
	I:REAL;
	D:REAL;
	Y_manual:REAL;
	Y_offset:REAL;
	Y_min:REAL;
	Y_max:REAL;
	manual:BOOL;
	reset:BOOL;
END_VAR
actual := set.actual;
set_point := set.set_point;
P := set.P;
I := set.I;
D := set.D;
Y_manual := set.Y_manual;
Y_offset := set.Y_offset;
Y_min := set.Y_min;
Y_max := set.Y_max;
manual := set.manual;
reset := set.reset;
END_FUNCTION_BLOCK

(* POU single_mode/Single, ST *)
FUNCTION_BLOCK Single
(* Function block implementation single mode. *)

VAR_INPUT
    enable: BOOL; (* Enable single mode *)
    pivot_pump: INT; (* pivot pump *)
    info_invertor_drive1: classInfoInvertorDrive;
    info_invertor_drive2: classInfoInvertorDrive;
    info_invertor_drive3: classInfoInvertorDrive;
    info_invertor_drive4: classInfoInvertorDrive;
    info_invertor_drive5: classInfoInvertorDrive;
    info_invertor_drive6: classInfoInvertorDrive;
    info_invertor_drive7: classInfoInvertorDrive;
    info_invertor_drive8: classInfoInvertorDrive;
END_VAR

VAR_OUTPUT
    info_single: classInfoSingle; (* info mode *)
END_VAR

VAR
    pivot: INT;
    pumps: ARRAY[1..8] OF BOOL;
END_VAR
pumps[1] := get_active(info_invertor_drive1);
pumps[2] := get_active(info_invertor_drive2);
pumps[3] := get_active(info_invertor_drive3);
pumps[4] := get_active(info_invertor_drive4);
pumps[5] := get_active(info_invertor_drive5);
pumps[6] := get_active(info_invertor_drive6);
pumps[7] := get_active(info_invertor_drive7);
pumps[8] := get_active(info_invertor_drive8);

pivot := pivot_pump;
IF pivot = 0 THEN
	enable := FALSE;
    info_single.error_code:=8;
END_IF;

IF enable THEN
    IF pumps[pivot] THEN
        info_single.pivot_pump := pivot;
        info_single.start_pump := pumps[pivot];
        info_single.error_code := 0;
        info_single.message := 'Select pump in work'; (* Выбранный насос в работе. *)
    ELSE
        info_single.pivot_pump := -8;
        info_single.start_pump := FALSE;
        info_single.error_code := 6;
        info_single.message := 'Select pump is not active!'; (* Выбранный насос не активен! *)
    END_IF;
      
ELSE
    info_single.pivot_pump := -8;
    info_single.start_pump := FALSE;
    info_single.error_code := 8;
    info_single.message := 'Single mode is not activate'; (* Режим работы одного насоса не активен. *)
END_IF;
END_FUNCTION_BLOCK

(* POU Invertor_Drive/get_active, ST *)
FUNCTION get_active : BOOL

VAR_INPUT
	info_invertor_drive:classInfoInvertorDrive;
END_VAR
get_active:=info_invertor_drive.active;
END_FUNCTION

(* POU cycle_mode/cycle, ST *)
FUNCTION_BLOCK cycle
(* Function block implementation cycle mode. *)

VAR_INPUT
	enable:BOOL;
	set_timer:TIME;
	info_invertor_drive1: classInfoInvertorDrive;
    info_invertor_drive2: classInfoInvertorDrive;
    info_invertor_drive3: classInfoInvertorDrive;
    info_invertor_drive4: classInfoInvertorDrive;
    info_invertor_drive5: classInfoInvertorDrive;
    info_invertor_drive6: classInfoInvertorDrive;
    info_invertor_drive7: classInfoInvertorDrive;
    info_invertor_drive8: classInfoInvertorDrive;
	END_VAR

VAR_OUTPUT
	info_cycle:classInfoCycle;
END_VAR
VAR
	pumps: ARRAY [1..8] OF BOOL;
	i: INT := 8;
	start_timer: TIME:=t#0ms;
	start_delay:TON;
	in: BOOL;

	working_time:TIME;
	Q:BOOL;
	n: INT;
END_VAR
pumps[1] := get_active(info_invertor_drive1);
pumps[2] := get_active(info_invertor_drive2);
pumps[3] := get_active(info_invertor_drive3);
pumps[4] := get_active(info_invertor_drive4);
pumps[5] := get_active(info_invertor_drive5);
pumps[6] := get_active(info_invertor_drive6);
pumps[7] := get_active(info_invertor_drive7);
pumps[8] := get_active(info_invertor_drive8);

n:=i;

IF pumps[i] = FALSE THEN
	i := i + 1;
END_IF;

IF  start_timer = t#0ms THEN
	start_timer := get_systime();
	in := TRUE;
END_IF;

working_time := work_time(start_timer);


IF working_time >= set_timer THEN
	in := FALSE;
	i := i + 1;
	start_timer := t#0ms;
END_IF;

start_delay(IN:=in, PT:=t#3s);
Q := start_delay.Q;

IF i > 8 THEN
	i := 1;
END_IF;

IF enable THEN
	info_cycle.working_time := working_time;
	info_cycle.run_timer := Q;
	info_cycle.pump_number := n;
ELSE
	info_cycle.working_time := T#0s;
	info_cycle.run_timer := FALSE;
	info_cycle.pump_number := 1;
	start_timer := t#0s;
END_IF;
info_cycle.error_code := 0;
END_FUNCTION_BLOCK

(* POU cycle_mode/get_systime, ST *)
FUNCTION get_systime : TIME

VAR_INPUT
END_VAR
get_systime:=TIME();
END_FUNCTION

(* POU cycle_mode/work_time, ST *)
FUNCTION work_time : TIME

VAR_INPUT
	start:TIME;
END_VAR
work_time:=TIME() - start;
END_FUNCTION

(* POU cascade_mode/cascade, ST *)
FUNCTION_BLOCK cascade
(* Functional block implementation cascade mode. *)
VAR_INPUT
	enable:BOOL;
	set_pressure:REAL;
	in_pressure: REAL;
	pivot_pump: INT;
	delay_on:TIME := t#30s;
	delay_off:TIME := t#30s;
    
	info_invertor_drive1: classInfoInvertorDrive;
    info_invertor_drive2: classInfoInvertorDrive;
    info_invertor_drive3: classInfoInvertorDrive;
    info_invertor_drive4: classInfoInvertorDrive;
    info_invertor_drive5: classInfoInvertorDrive;
    info_invertor_drive6: classInfoInvertorDrive;
    info_invertor_drive7: classInfoInvertorDrive;
    info_invertor_drive8: classInfoInvertorDrive;
END_VAR

VAR_OUTPUT
	info_cascade:classInfoCascade;
END_VAR

VAR
	pumps: ARRAY [1..8] OF BOOL;
	cascade_pumps: ARRAY [1..8] OF classInfoCascadePump;
	pivot: INT;
	i: INT:=1;
	error_message: STRING(79):= 'NOT GOOD';
	start_time: TIME:=t#0s;
	work_time: TIME;
	len_pumps: INT;
	index_active_pumps:ARRAY [1..8] OF INT;
	len_active_pumps: INT;
	index_pivot: INT;
	histeresys: REAL := 0.2 (* histeresys set pressure *);
	error_code:WORD;
END_VAR
pivot := pivot_pump;

IF pivot = 0 THEN
	check_pivot;
ELSE
    check_active_pumps;
END_IF;

IF len_active_pumps > 1  AND index_pivot <> 0 THEN
    cascade_on;
ELSIF len_active_pumps = 1 AND index_pivot <> 0 THEN
    i := index_pivot;
	error_code := 4;
    error_message := 'cascade mode excpected more one active pumps, but got less';
ELSIF index_pivot = 0 THEN
	error_code := 5;
	error_message := 'pivot pump not active';
END_IF;

get_info_message;
END_FUNCTION_BLOCK
ACTION cascade_on:
error_code := 0;
error_message := 'GOOD';

(* inspect bounds array. *)

IF i = 1 AND i = index_pivot THEN
	i := pivot + 1;
ELSIF i = len_active_pumps AND  i = index_pivot THEN
	i := len_active_pumps - 1;
END_IF;

(* start pivot pump. *)
IF INT_TO_BOOL(index_pivot) THEN
	cascade_pumps[pivot].cascade_pump := TRUE;
END_IF;

IF start_time = t#0s THEN
	start_time := TIME();
END_IF;


IF in_pressure < (set_pressure - histeresys) THEN
	work_time := TIME() - start_time;
	IF work_time >= delay_on THEN
		IF i = index_pivot AND index_pivot < len_active_pumps THEN
			i := i + 1;
		END_IF;
		cascade_pumps[index_active_pumps[i]].cascade_pump := TRUE;
		i := i + 1;
		start_time := t#0s;
	END_IF;
ELSIF in_pressure > (set_pressure + histeresys) THEN
	work_time := TIME() - start_time;
	IF work_time >= delay_off THEN
		IF i = index_pivot AND index_pivot > 1 THEN
			i := i - 1;
		END_IF;
		cascade_pumps[index_active_pumps[i]].cascade_pump := FALSE;
		i := i - 1;
		start_time := t#0s;
	END_IF;
END_IF;

IF i > len_active_pumps  THEN
	i := len_active_pumps;
ELSIF i < 1 THEN
	i := 1;
END_IF;
END_ACTION
ACTION check_active_pumps:
pumps[1] := get_active(info_invertor_drive1);
pumps[2] := get_active(info_invertor_drive2);
pumps[3] := get_active(info_invertor_drive3);
pumps[4] := get_active(info_invertor_drive4);
pumps[5] := get_active(info_invertor_drive5);
pumps[6] := get_active(info_invertor_drive6);
pumps[7] := get_active(info_invertor_drive7);
pumps[8] := get_active(info_invertor_drive8);

len_pumps := len_bool_array(pumps);  (* get en input pumps array. *)
index_active_pumps := index_bool_array(pumps);  (* get indexes active pumps. *)
len_active_pumps := len_int_array(index_active_pumps);  (* get len active pumps. *)

index_pivot := index_element_in_int_array(pivot, index_active_pumps); (* get index pivot.*)
END_ACTION
ACTION check_pivot:
error_code := 3;
error_message := 'pivot pump not excpect int more 0.';
END_ACTION
ACTION get_info_message:
IF enable AND error_message = 'GOOD' THEN
	info_cascade.pivot := pivot;
	info_cascade.error_message := error_message;
	info_cascade.cascade_pump1 := cascade_pumps[1];
	info_cascade.cascade_pump2 := cascade_pumps[2];
	info_cascade.cascade_pump3 := cascade_pumps[3];
	info_cascade.cascade_pump4 := cascade_pumps[4];
	info_cascade.cascade_pump5 := cascade_pumps[5];
	info_cascade.cascade_pump6 := cascade_pumps[6];
	info_cascade.cascade_pump7 := cascade_pumps[7];
	info_cascade.cascade_pump8 := cascade_pumps[8];
	info_cascade.error_code := error_code;
ELSE
	info_cascade.pivot := index_pivot;
	info_cascade.error_code := error_code;
	info_cascade.error_message := error_message;
	cascade_pumps[1].cascade_pump := FALSE;
	cascade_pumps[2].cascade_pump := FALSE;
	cascade_pumps[3].cascade_pump := FALSE;
	cascade_pumps[4].cascade_pump := FALSE;
	cascade_pumps[5].cascade_pump := FALSE;
	cascade_pumps[6].cascade_pump := FALSE;
	cascade_pumps[7].cascade_pump := FALSE;
	cascade_pumps[8].cascade_pump := FALSE;
	info_cascade.cascade_pump1 := cascade_pumps[1];
	info_cascade.cascade_pump2 := cascade_pumps[2];
	info_cascade.cascade_pump3 := cascade_pumps[3];
	info_cascade.cascade_pump4 := cascade_pumps[4];
	info_cascade.cascade_pump5 := cascade_pumps[5];
	info_cascade.cascade_pump6 := cascade_pumps[6];
	info_cascade.cascade_pump7 := cascade_pumps[7];
	info_cascade.cascade_pump8 := cascade_pumps[8];
END_IF;
END_ACTION

(* POU function/methods_8_array/len_bool_array, ST *)
FUNCTION len_bool_array : INT

VAR_INPUT
	list: ARRAY [1..8] OF BOOL;
END_VAR

VAR
	size: INT := 8;
	cnt:INT := 0;
	i: INT;
END_VAR
FOR i := 1 TO size DO
	IF list[i] THEN
		cnt := cnt + 1;
	END_IF;
END_FOR;

IF i > 8 THEN
	i := 1;
END_IF;

len_bool_array := cnt;
END_FUNCTION

(* POU function/methods_8_array/index_bool_array, ST *)
FUNCTION index_bool_array : ARRAY [1..8] OF INT

VAR_INPUT
	list:ARRAY [1..8] OF BOOL;
END_VAR

VAR
	size:INT := 8;
	i: INT;
	cnt:INT := 1;
	index:ARRAY [1..8] OF INT := 8(0);
END_VAR
FOR i:= 1 TO size DO
	IF list[i] THEN
		index[cnt] := i;
		cnt := cnt + 1;
	END_IF;
END_FOR;

index_bool_array := index;
END_FUNCTION

(* POU function/methods_8_array/len_int_array, ST *)
FUNCTION len_int_array : INT

VAR_INPUT
	list: ARRAY [1..8] OF INT;
END_VAR

VAR
	size: INT:=8;
	cnt:INT:=0;
	i: INT;
END_VAR
FOR i:=1 TO size DO
	IF INT_TO_BOOL(list[i]) THEN
		cnt:=cnt + 1;
	END_IF;
END_FOR;

IF i > 8 THEN
	i:=1;
END_IF;

len_int_array:=cnt;
END_FUNCTION

(* POU function/methods_8_array/index_element_in_int_array, ST *)
FUNCTION index_element_in_int_array : INT

VAR_INPUT
	element:INT;
	list:ARRAY [1..8] OF  INT;
END_VAR

VAR
	size: INT := 8;
	i: INT;
	index: INT := 1;
END_VAR
IF element_in_int_array(element, list) THEN
	FOR i := 1 TO size DO
		IF list[i]=element THEN
			index := i;
			i := 8;
		END_IF;
	END_FOR;
	index_element_in_int_array := index;
ELSE
	index_element_in_int_array := 0;
END_IF;
END_FUNCTION

(* POU function/methods_8_array/element_in_int_array, ST *)
FUNCTION element_in_int_array : BOOL

VAR_INPUT
	element:INT;
	list: ARRAY [1..8] OF INT;
END_VAR

VAR
	size: INT := 8;
	i: INT;
	is_true:BOOL := FALSE;
END_VAR
FOR i := 1 TO size DO
	IF list[i]=element THEN
		is_true := TRUE;
	END_IF;
END_FOR;

element_in_int_array := is_true;
END_FUNCTION

(* POU mode_selector/Cascade_Cycle_Selector, ST *)
FUNCTION_BLOCK Cascade_Cycle_Selector
(* Function block implementation working mode selector. *)

VAR_INPUT
    cascade: BOOL; (* enable/disable *)
    cycle: BOOL; (* enable/disable *)
    single: BOOL; (* enable/disable *)
    info_single: classInfoSingle;
    info_cycle: classInfoCycle;
    info_cascade: classInfoCascade;
END_VAR

VAR_OUTPUT
    mode_selector_error: WORD;
    start_pump1: BOOL := FALSE;
    start_pump2: BOOL := FALSE;
    start_pump3: BOOL := FALSE;
    start_pump4: BOOL := FALSE;
    start_pump5: BOOL := FALSE;
    start_pump6: BOOL := FALSE;
    start_pump7: BOOL := FALSE;
    start_pump8: BOOL := FALSE;
END_VAR

VAR
    message: STRING(79);
    flag_mode: INT;
	error_code: WORD;
END_VAR
IF cascade AND NOT cycle AND NOT single THEN
    flag_mode := 2;
    message := 'Cascade mode selected'; (* Выбран каскадный режим работы. *)
ELSIF cycle AND NOT cascade AND NOT single THEN
    flag_mode := 1;
    message := 'Cycle mode selected'; (* Выбран циклический режим работы *)
ELSIF single AND NOT cycle AND NOT cascade THEN
    flag_mode := 0;
    message := 'Single mode selected'; (* Выбран режим работы одного насоса *) 
ELSE
    flag_mode := -1;
    error_code := 7;
    message := 'Select any one working mode!'; (* Выберите один режим работы! *)
END_IF;

IF flag_mode = 0 THEN
    start_pump1 := get_pump_in_single(info_single, 1);
    start_pump2 := get_pump_in_single(info_single, 2);
    start_pump3 := get_pump_in_single(info_single, 3);
    start_pump4 := get_pump_in_single(info_single, 4);
    start_pump5 := get_pump_in_single(info_single, 5);
    start_pump6 := get_pump_in_single(info_single, 6);
    start_pump7 := get_pump_in_single(info_single, 7);
    start_pump8 := get_pump_in_single(info_single, 8);
    mode_selector_error := info_single.error_code;
ELSIF flag_mode = 1 THEN
    start_pump1 := get_pump_in_cycle(info_cycle, 1);
    start_pump2 := get_pump_in_cycle(info_cycle, 2);
    start_pump3 := get_pump_in_cycle(info_cycle, 3);
    start_pump4 := get_pump_in_cycle(info_cycle, 4);
    start_pump5 := get_pump_in_cycle(info_cycle, 5);
    start_pump6 := get_pump_in_cycle(info_cycle, 6);
    start_pump7 := get_pump_in_cycle(info_cycle, 7);
    start_pump8 := get_pump_in_cycle(info_cycle, 8);
    mode_selector_error := info_cycle.error_code;
ELSIF flag_mode = 2 THEN
    start_pump1 := get_pump_in_cascade(info_cascade, 1);
    start_pump2 := get_pump_in_cascade(info_cascade, 2);
    start_pump3 := get_pump_in_cascade(info_cascade, 3);
    start_pump4 := get_pump_in_cascade(info_cascade, 4);
    start_pump5 := get_pump_in_cascade(info_cascade, 5);
    start_pump6 := get_pump_in_cascade(info_cascade, 6);
    start_pump7 := get_pump_in_cascade(info_cascade, 7);
    start_pump8 := get_pump_in_cascade(info_cascade, 8);
    mode_selector_error := info_cascade.error_code;
ELSE
    start_pump1 := FALSE;
    start_pump2 := FALSE;
    start_pump3 := FALSE;
    start_pump4 := FALSE;
    start_pump5 := FALSE;
    start_pump6 := FALSE;
    start_pump7 := FALSE;
    start_pump8 := FALSE;
    mode_selector_error := error_code;
END_IF;
END_FUNCTION_BLOCK

(* POU single_mode/get_pump_in_single, ST *)
FUNCTION get_pump_in_single : BOOL
(* Function get status pump in information single mode *)

VAR_INPUT
    info_single: classInfoSingle;
    pump_number: INT;
END_VAR
IF pump_number = info_single.pivot_pump THEN
    get_pump_in_single := info_single.start_pump;
ELSE
    get_pump_in_single := FALSE;
END_IF;
END_FUNCTION

(* POU cycle_mode/get_pump_in_cycle, ST *)
FUNCTION get_pump_in_cycle : BOOL (*ï¿½ï¿½ï¿½ï¿½ï¿½ï¿½ï¿½ ï¿½ï¿½ï¿½ï¿½ï¿½ï¿½ï¿½ï¿½ï¿½ï¿½ï¿½ï¿½ ï¿½ï¿½ï¿½ï¿½ ï¿½ï¿½ï¿½ï¿½ï¿½ï¿½ ï¿½ï¿½ï¿½ï¿½ï¿½ï¿½ï¿½ï¿½ï¿½ï¿½ ï¿½ï¿½ï¿½ï¿½ï¿½ï¿½ *)

VAR_INPUT
	info_cycle:classInfoCycle;
	pump_number:SINT;
END_VAR
IF pump_number=info_cycle.pump_number THEN
	get_pump_in_cycle:=info_cycle.run_timer;
ELSE
	get_pump_in_cycle:=FALSE;
END_IF;
END_FUNCTION

(* POU cascade_mode/get_pump_in_cascade, ST *)
FUNCTION get_pump_in_cascade : BOOL

VAR_INPUT
	info:classInfoCascade;
	number_pump:INT;
END_VAR

VAR
	pumps:ARRAY[1..8] OF classInfoCascadePump;
END_VAR
IF info.pivot = number_pump THEN
	get_pump_in_cascade:=TRUE;
ELSE
	pumps[1]:=info.cascade_pump1;
	pumps[2]:=info.cascade_pump2;
	pumps[3]:=info.cascade_pump3;
	pumps[4]:=info.cascade_pump4;
	pumps[5]:=info.cascade_pump5;
	pumps[6]:=info.cascade_pump6;
	pumps[7]:=info.cascade_pump7;
	pumps[8]:=info.cascade_pump8;

	get_pump_in_cascade:=pumps[number_pump].cascade_pump;
END_IF;
END_FUNCTION

(* POU DanfossKPI/Kpi, ST *)
FUNCTION_BLOCK Kpi

VAR_INPUT
	input:BOOL;  (* ï¿½ï¿½ï¿½ï¿½ï¿½ï¿½ï¿½ï¿½ ï¿½ï¿½ ï¿½ï¿½ï¿½ï¿½ï¿½ *)
END_VAR

VAR_OUTPUT
	NC:BOOL; (* normal close �2 *)
	NO:BOOL; (* normal open �4 *)
END_VAR

VAR
END_VAR
NC:=NOT input;
NO:=input;
END_FUNCTION_BLOCK

(* POU Alarm_manager_error/ALARM_MANAGER, ST *)
FUNCTION_BLOCK ALARM_MANAGER
(* Function block handle alarm. *)

VAR_INPUT
    low_pressure_input: BOOL;
    high_pressure_out: BOOL;
    external_alarm_invertor_drive_code: WORD;
    input_pressure_error_code: WORD;
    out_pressure_error_code: WORD;
    mode_selector_error: WORD;
END_VAR

VAR_OUTPUT
    alarm_on: BOOL := TRUE;
    error_code_alarm: WORD;
    error_message: STRING(79);
END_VAR
IF low_pressure_input THEN
    error_code_alarm := 1;
ELSIF high_pressure_out THEN
    error_code_alarm := 2;
ELSIF external_alarm_invertor_drive_code > 0 THEN
    error_code_alarm := external_alarm_invertor_drive_code;
ELSIF input_pressure_error_code > 0 THEN
    error_code_alarm := input_pressure_error_code;
ELSIF out_pressure_error_code > 0 THEN
    error_code_alarm := input_pressure_error_code;
ELSIF mode_selector_error > 0 THEN
    error_code_alarm := mode_selector_error;
ELSE
    error_code_alarm := 0;
END_IF;

IF error_code_alarm <> 0 THEN
    alarm_on := TRUE;
    error_message := get_alarm_message(error_code_alarm);
ELSE
    alarm_on := FALSE;
END_IF;
END_FUNCTION_BLOCK

(* POU Alarm_manager_error/get_alarm_message, ST *)
FUNCTION get_alarm_message : STRING(79)
(* Function return message alarm of error_code *)

VAR_INPUT
    code_error: WORD;
END_VAR

VAR
    error_message: STRING(79);
END_VAR
IF code_error = 0
	THEN error_message := 'Measure good.'; (* Измерение успешно. *)
ELSIF code_error = 1
    THEN error_message := 'low input pressure!'; (* Низкое давление на выходе. *)
ELSIF code_error = 2 
    THEN error_message := 'high output pressure!'; (* Превышение давления на выходе. *)
ELSIF code_error = 3
    THEN error_message := 'Pivot cascade pump not expected int more 0!'; (* Опорный насос не может быть 0 *)
ELSIF code_error = 4
    THEN error_message := 'Cascade mode excpected more one active pumps, but got less!'; (* В каскадном режиме должно быть больше одного активного насоса. *)
ELSIF code_error = 5
    THEN error_message := 'Cascade pivot pump not active!'; (* Опорный насос в каскадном режиме не активен. *)
ELSIF code_error = 6
    THEN error_message := 'Single mode select pump is not active!'; (* Опорный насос в одиночном режиме на активен *)
ELSIF code_error = 7
    THEN error_message := 'Select any one working mode!'; (* Выберите только один режим работы станции. *)
ELSIF code_error = 8
    THEN error_message := 'External alarm invertor drive 1'; (* Внешняя авария на частотном преобразователе 1. *)
ELSIF code_error = 9
    THEN error_message := 'External alarm invertor drive 2'; (* Внешняя авария на частотном преобразователе 2. *)
ELSIF code_error = 10
    THEN error_message := 'External alarm invertor drive 3'; (* Внешняя авария на частотном преобразователе 3. *)
ELSIF code_error = 11
    THEN error_message := 'External alarm invertor drive 4'; (* Внешняя авария на частотном преобразователе 4. *)
ELSIF code_error = 12
    THEN error_message := 'External alarm invertor drive 5'; (* Внешняя авария на частотном преобразователе 5. *)
ELSIF code_error = 13
    THEN error_message := 'External alarm invertor drive 6'; (* Внешняя авария на частотном преобразователе 6. *)
ELSIF code_error = 14
    THEN error_message := 'External alarm invertor drive 7'; (* Внешняя авария на частотном преобразователе 7. *)
ELSIF code_error = 15
    THEN error_message := 'External alarm invertor drive 8'; (* Внешняя авария на частотном преобразователе 8. *)
ELSIF code_error = 61440
	THEN error_message := 'Value bad!'; (* Значение заведомо неверно. *)
ELSIF code_error = 61446
	THEN error_message := 'Data info not complete! Wait first measuring.'; (* Данные не готовы. Ждите результатов первого измерения. *)
ELSIF code_error = 61447
	THEN error_message := 'Sensor off.'; (* Датчик отключен. *)
ELSIF code_error = 61448
	THEN error_message := 'Temperature free ends of termosensor high.'; (* Велика температура свободных концов ТП. *)
ELSIF code_error = 61449
	THEN error_message := 'Temperature free ends of termosensor low.'; (* Мала температура свободных концов ТП. *)
ELSIF code_error = 61450
	THEN error_message := 'Measured value too more.'; (* Измеренное значение слишком велико. *)
ELSIF code_error = 61451
	THEN error_message := 'Measured value too less.'; (* Измеренное значение слишком мало. *)
ELSIF code_error = 61452
	THEN error_message := 'Short circuit of sensor.'; (* Короткое замыкание датчика. *)
ELSIF code_error = 61453
	THEN error_message := 'Sensor breaking.'; (* Обрыв датчика. *)
ELSIF code_error = 61454
	THEN error_message := 'Failure connection with DAC.'; (* Отсутствие связи с АЦП. *)
ELSIF code_error = 61455
	THEN error_message := 'Uncorrect calibrate rate.'; (* Некорректный калибровочный коэффициент. *)
ELSE
	error_message := 'Error not Found';
END_IF

get_alarm_message := error_message;
    
END_FUNCTION

(* POU Alarm_manager_error/external_alarm_invertor_drive, ST *)
FUNCTION_BLOCK external_alarm_invertor_drive
(* Function block return code error external alarm of invertor drives in PLC110-32m2 *)

VAR_INPUT
    status_inputs: classPLC32m2StatusInputs;
    number_di_alarm_id1: INT := 0;
    number_di_alarm_id2: INT := 0;
    number_di_alarm_id3: INT := 0;
    number_di_alarm_id4: INT := 0;
    number_di_alarm_id5: INT := 0;
    number_di_alarm_id6: INT := 0;
    number_di_alarm_id7: INT := 0;
    number_di_alarm_id8: INT := 0;
END_VAR

VAR_OUTPUT
    error_code_alarm: WORD;
END_VAR

VAR
    check_alarm: INT;
    error_code: WORD;
    i: INT;
    number_di_alarm: ARRAY [1..8] OF INT;
    pump_alarm: ARRAY [1..8] OF BOOL;
    index_alarm: ARRAY [1..8] OF INT;
END_VAR
number_di_alarm[1] := number_di_alarm_id1;
number_di_alarm[2] := number_di_alarm_id2;
number_di_alarm[3] := number_di_alarm_id3;
number_di_alarm[4] := number_di_alarm_id4;
number_di_alarm[5] := number_di_alarm_id5;
number_di_alarm[6] := number_di_alarm_id6;
number_di_alarm[7] := number_di_alarm_id7;
number_di_alarm[8] := number_di_alarm_id8;

FOR i := 1 TO 8 DO
    IF number_di_alarm[i] > 0 THEN
        pump_alarm[i] := get_di(number_di_alarm[i], status_inputs);
    ELSE
        pump_alarm[i] := FALSE;
    END_IF;
END_FOR;

check_alarm := len_bool_array(pump_alarm);
IF check_alarm > 0  THEN
    index_alarm := index_bool_array(pump_alarm);
    error_code := 7 + index_alarm[1];
ELSE
    error_code := check_alarm;
END_IF;

error_code_alarm := error_code;
END_FUNCTION_BLOCK

(* POU PLC110_32/get_di, ST *)
FUNCTION get_di : BOOL

VAR_INPUT
	input_number:INT;
	status_inputs:classPLC32m2StatusInputs;
END_VAR

VAR
	in_f:classDiscreteInputByte;
	in_s:classDiscreteInputByte;
	di_list:ARRAY[1..17] OF BOOL;
END_VAR
in_f:=status_inputs.discrete_inputs.first_byte;
in_s:=status_inputs.discrete_inputs.second_byte;

di_list[1]:=in_f.Bit1;
di_list[2]:=in_f.Bit2;
di_list[3]:=in_f.Bit3;
di_list[4]:=in_f.Bit4;
di_list[5]:=in_f.Bit5;
di_list[6]:=in_f.Bit6;
di_list[7]:=in_f.Bit7;
di_list[8]:=in_f.Bit8;

di_list[9]:=in_s.Bit1;
di_list[10]:=in_s.Bit2;
di_list[11]:=in_s.Bit3;
di_list[12]:=in_s.Bit4;
di_list[13]:=in_s.Bit5;
di_list[14]:=in_s.Bit6;
di_list[15]:=in_s.Bit7;
di_list[16]:=in_s.Bit8;

get_di:=di_list[input_number];
END_FUNCTION

(* POU PressureSensor_4_20ma/SetCurrentSensorPressure_4_20, ST *)
FUNCTION_BLOCK SetCurrentSensorPressure_4_20

VAR_INPUT
	min_measure_range:REAL:=0;
	max_measure_range:REAL:=16;
	min_current_range:REAL:=4;
	max_current_range:REAL:=20;
END_VAR

VAR_OUTPUT
	sensor_params:classSetPressureSensor4_20;
END_VAR
sensor_params.min_measure_range := min_measure_range;
sensor_params.max_measure_range := max_measure_range;
sensor_params.min_current_range := min_current_range;
sensor_params.max_current_range := max_current_range;
END_FUNCTION_BLOCK

(* POU Invertor_Drive/get_aout_current_in_info, ST *)
FUNCTION get_aout_current_in_info : REAL

VAR_INPUT
	info_invertor_drive:classInfoInvertorDrive;
END_VAR
get_aout_current_in_info:=info_invertor_drive.aout_frequency;
END_FUNCTION

(* POU Invertor_Drive/get_run_in_info, ST *)
FUNCTION get_run_in_info : BOOL

VAR_INPUT
	info_invertor_drive:classInfoInvertorDrive;
END_VAR
get_run_in_info:=info_invertor_drive.run ;
END_FUNCTION

(* POU Invertor_Drive/get_reset_faults, ST *)
FUNCTION get_reset_faults : BOOL

VAR_INPUT
    info: classInfoInvertorDrive; (* Comment *)
END_VAR
get_reset_faults := info.reset_fault;
END_FUNCTION

(* POU MB110_8.A/get_channel_current_value, ST *)
FUNCTION get_channel_current_value : REAL
(* ï¿½ï¿½ï¿½ï¿½ï¿½ï¿½ï¿½ ï¿½ï¿½ï¿½ï¿½ï¿½ï¿½ï¿½ï¿½ï¿½ï¿½ï¿½ï¿½ï¿½ InfoMessage ï¿½ï¿½ AnalogInputsModule  ï¿½ ï¿½ï¿½ï¿½ï¿½ï¿½ï¿½ï¿½ ï¿½ï¿½ ï¿½ï¿½ï¿½ï¿½ï¿½ï¿½ï¿½ ï¿½ï¿½ï¿½ï¿½ï¿½ï¿½ ï¿½ï¿½ï¿½ï¿½ï¿½ï¿½ï¿½ï¿½ ï¿½ï¿½ï¿½ï¿½ *)

VAR_INPUT
	ch_number:INT;
	Ain_info:classInfoAnalogInputModule;
END_VAR

VAR
	list_value : ARRAY [1..8] OF REAL;
END_VAR
list_value[1] := Ain_info.channel1.current_value;
list_value[2] := Ain_info.channel2.current_value;
list_value[3] := Ain_info.channel3.current_value;
list_value[4] := Ain_info.channel4.current_value;
list_value[5] := Ain_info.channel5.current_value;
list_value[6] := Ain_info.channel6.current_value;
list_value[7] := Ain_info.channel7.current_value;
list_value[8] := Ain_info.channel8.current_value;

get_channel_current_value := list_value[ch_number];
END_FUNCTION

(* POU function/hms_to_time, ST *)
FUNCTION hms_to_time : TIME
VAR_INPUT
	hours: WORD;
	minutes: WORD;
	seconds: WORD;
END_VAR
VAR
	MILLISECONDS_IN_HOUR: DWORD := 3600000;
	MILLISECONDS_IN_MINUTE: DWORD := 60000;
	MILLISECONDS_IN_SECOND: DWORD := 1000;
END_VAR
hms_to_time := DWORD_TO_TIME(
    (WORD_TO_DWORD(hours) * MILLISECONDS_IN_HOUR)
    + (WORD_TO_DWORD(minutes) * MILLISECONDS_IN_MINUTE)
    + (WORD_TO_DWORD(seconds) * MILLISECONDS_IN_SECOND)
);
END_FUNCTION

(* POU cascade_mode/get_auto_in_cascade, ST *)
FUNCTION get_auto_in_cascade : BOOL

VAR_INPUT
	info:classInfoCascade;
	number_pump:INT;
END_VAR
IF info.pivot=number_pump THEN
	get_auto_in_cascade:=TRUE;
ELSE
	get_auto_in_cascade:=FALSE;
END_IF;
END_FUNCTION

(* POU Invertor_Drive/get_frequency_in_info, ST *)
FUNCTION get_frequency_in_info : REAL
VAR_INPUT
	info_invertor_drive:classInfoInvertorDrive;
END_VAR
VAR
END_VAR
get_frequency_in_info:=info_invertor_drive.frequency;
END_FUNCTION

(* POU PLC110_32/get_fdi, ST *)
FUNCTION get_fdi : BOOL
(* ï¿½ï¿½ï¿½ï¿½ï¿½ï¿½ï¿½ï¿½ï¿½ï¿½ï¿½ï¿½ï¿½ ï¿½ï¿½ ï¿½ï¿½ï¿½ï¿½ï¿½ï¿½ï¿½ ï¿½ï¿½ï¿½ï¿½ï¿½ï¿½ ï¿½ï¿½ï¿½ï¿½ï¿½ï¿½ ï¿½ï¿½ï¿½ï¿½ï¿½ï¿½ï¿½ï¿½ï¿½ FDI *)
VAR_INPUT
	num:INT;
	status_inputs:classPLC32m2StatusInputs;
END_VAR

VAR
	fdi_list:ARRAY [1..2] OF BOOL;
END_VAR
fdi_list[1]:=status_inputs.fast_inputs.Bit1;
fdi_list[2]:=status_inputs.fast_inputs.Bit2;

get_fdi:=fdi_list[num];
END_FUNCTION
